  PROC DrawPart265()
    MoveL Offs(pOrigin,121.94,113.28,0.00),v40,z0,tPen\WObj:=wPaper;
    MoveL Offs(pOrigin,121.19,112.53,0.00),v40,z0,tPen\WObj:=wPaper;
    MoveL Offs(pOrigin,121.43,111.79,0.00),v40,z0,tPen\WObj:=wPaper;
    MoveL Offs(pOrigin,119.78,113.44,0.00),v40,z0,tPen\WObj:=wPaper;
    MoveL Offs(pOrigin,120.15,112.97,0.00),v40,z0,tPen\WObj:=wPaper;
    MoveL Offs(pOrigin,117.74,110.57,0.00),v40,z0,tPen\WObj:=wPaper;
    MoveL Offs(pOrigin,117.82,111.25,0.00),v40,z0,tPen\WObj:=wPaper;
    MoveL Offs(pOrigin,118.68,111.32,0.00),v40,z0,tPen\WObj:=wPaper;
    MoveL Offs(pOrigin,119.31,112.10,0.00),v40,z0,tPen\WObj:=wPaper;
    MoveL Offs(pOrigin,120.38,112.60,0.00),v40,z0,tPen\WObj:=wPaper;
    MoveL Offs(pOrigin,127.81,114.65,0.00),v40,fine,tPen\WObj:=wPaper;
    MoveL Offs(pOrigin,127.81,114.65,6.00),v60,z5,tPen\WObj:=wPaper;
    MoveL Offs(pOrigin,126.82,113.87,6.00),vTravel,z5,tPen\WObj:=wPaper;
    MoveL Offs(pOrigin,126.82,113.87,0.00),v60,z0,tPen\WObj:=wPaper;
    MoveL Offs(pOrigin,125.91,114.77,0.00),v40,fine,tPen\WObj:=wPaper;
    MoveL Offs(pOrigin,125.91,114.77,6.00),v60,z5,tPen\WObj:=wPaper;
    MoveL Offs(pOrigin,125.77,113.43,6.00),vTravel,z5,tPen\WObj:=wPaper;
    MoveL Offs(pOrigin,125.77,113.43,0.00),v60,z0,tPen\WObj:=wPaper;
    MoveL Offs(pOrigin,124.57,114.63,0.00),v40,fine,tPen\WObj:=wPaper;
    MoveL Offs(pOrigin,124.57,114.63,6.00),v60,z5,tPen\WObj:=wPaper;
    MoveL Offs(pOrigin,123.37,114.33,6.00),vTravel,z5,tPen\WObj:=wPaper;
    MoveL Offs(pOrigin,123.37,114.33,0.00),v60,z0,tPen\WObj:=wPaper;
    MoveL Offs(pOrigin,124.72,112.98,0.00),v40,fine,tPen\WObj:=wPaper;
    MoveL Offs(pOrigin,124.72,112.98,6.00),v60,z5,tPen\WObj:=wPaper;
    MoveL Offs(pOrigin,126.07,111.63,6.00),vTravel,z5,tPen\WObj:=wPaper;
    MoveL Offs(pOrigin,126.07,111.63,0.00),v60,z0,tPen\WObj:=wPaper;
    MoveL Offs(pOrigin,126.97,110.73,0.00),v40,fine,tPen\WObj:=wPaper;
    MoveL Offs(pOrigin,126.97,110.73,6.00),v60,z5,tPen\WObj:=wPaper;
    MoveL Offs(pOrigin,127.12,112.07,6.00),vTravel,z5,tPen\WObj:=wPaper;
    MoveL Offs(pOrigin,127.12,112.07,0.00),v60,z0,tPen\WObj:=wPaper;
    MoveL Offs(pOrigin,128.47,110.72,0.00),v40,fine,tPen\WObj:=wPaper;
    MoveL Offs(pOrigin,128.47,110.72,6.00),v60,z5,tPen\WObj:=wPaper;
    MoveL Offs(pOrigin,129.82,110.87,6.00),vTravel,z5,tPen\WObj:=wPaper;
    MoveL Offs(pOrigin,129.82,110.87,0.00),v60,z0,tPen\WObj:=wPaper;
    MoveL Offs(pOrigin,128.32,112.37,0.00),v40,fine,tPen\WObj:=wPaper;
    MoveL Offs(pOrigin,128.32,112.37,6.00),v60,z5,tPen\WObj:=wPaper;
    MoveL Offs(pOrigin,129.52,112.67,6.00),vTravel,z5,tPen\WObj:=wPaper;
    MoveL Offs(pOrigin,129.52,112.67,0.00),v60,z0,tPen\WObj:=wPaper;
    MoveL Offs(pOrigin,131.32,110.86,0.00),v40,fine,tPen\WObj:=wPaper;
    MoveL Offs(pOrigin,131.32,110.86,6.00),v60,z5,tPen\WObj:=wPaper;
    MoveL Offs(pOrigin,132.82,110.86,6.00),vTravel,z5,tPen\WObj:=wPaper;
    MoveL Offs(pOrigin,132.82,110.86,0.00),v60,z0,tPen\WObj:=wPaper;
    MoveL Offs(pOrigin,130.86,112.81,0.00),v40,fine,tPen\WObj:=wPaper;
    MoveL Offs(pOrigin,130.86,112.81,6.00),v60,z5,tPen\WObj:=wPaper;
    MoveL Offs(pOrigin,126.65,118.52,6.00),vTravel,z5,tPen\WObj:=wPaper;
    MoveL Offs(pOrigin,126.65,118.52,0.00),v60,z0,tPen\WObj:=wPaper;
    MoveL Offs(pOrigin,124.85,120.32,0.00),v40,z0,tPen\WObj:=wPaper;
    MoveL Offs(pOrigin,125.86,120.18,0.00),v40,z0,tPen\WObj:=wPaper;
    MoveL Offs(pOrigin,122.86,117.17,0.00),v40,z0,tPen\WObj:=wPaper;
    MoveL Offs(pOrigin,122.76,116.43,0.00),v40,z0,tPen\WObj:=wPaper;
    MoveL Offs(pOrigin,121.26,117.93,0.00),v40,z0,tPen\WObj:=wPaper;
    MoveL Offs(pOrigin,122.11,117.92,0.00),v40,z0,tPen\WObj:=wPaper;
    MoveL Offs(pOrigin,120.91,116.72,0.00),v40,z0,tPen\WObj:=wPaper;
    MoveL Offs(pOrigin,120.36,117.34,0.00),v40,z0,tPen\WObj:=wPaper;
    MoveL Offs(pOrigin,121.72,115.99,0.00),v40,z0,tPen\WObj:=wPaper;
    MoveL Offs(pOrigin,120.67,115.54,0.00),v40,z0,tPen\WObj:=wPaper;
    MoveL Offs(pOrigin,119.32,116.89,0.00),v40,z0,tPen\WObj:=wPaper;
    MoveL Offs(pOrigin,118.72,115.99,0.00),v40,z0,tPen\WObj:=wPaper;
    MoveL Offs(pOrigin,119.77,114.94,0.00),v40,fine,tPen\WObj:=wPaper;
    MoveL Offs(pOrigin,119.77,114.94,6.00),v60,z5,tPen\WObj:=wPaper;
    MoveL Offs(pOrigin,118.57,114.65,6.00),vTravel,z5,tPen\WObj:=wPaper;
    MoveL Offs(pOrigin,118.57,114.65,0.00),v60,z0,tPen\WObj:=wPaper;
    MoveL Offs(pOrigin,117.82,115.40,0.00),v40,fine,tPen\WObj:=wPaper;
    MoveL Offs(pOrigin,117.82,115.40,6.00),v60,z5,tPen\WObj:=wPaper;
    MoveL Offs(pOrigin,116.97,114.44,6.00),vTravel,z5,tPen\WObj:=wPaper;
    MoveL Offs(pOrigin,116.97,114.44,0.00),v60,z0,tPen\WObj:=wPaper;
    MoveL Offs(pOrigin,129.30,121.66,0.00),v40,z0,tPen\WObj:=wPaper;
    MoveL Offs(pOrigin,131.43,123.57,0.00),v40,z0,tPen\WObj:=wPaper;
    MoveL Offs(pOrigin,131.64,124.21,0.00),v40,fine,tPen\WObj:=wPaper;
    MoveL Offs(pOrigin,131.64,124.21,6.00),v60,z5,tPen\WObj:=wPaper;
    MoveL Offs(pOrigin,130.38,123.75,6.00),vTravel,z5,tPen\WObj:=wPaper;
    MoveL Offs(pOrigin,130.38,123.75,0.00),v60,z0,tPen\WObj:=wPaper;
    MoveL Offs(pOrigin,131.58,122.55,0.00),v40,z0,tPen\WObj:=wPaper;
    MoveL Offs(pOrigin,130.84,121.80,0.00),v40,z0,tPen\WObj:=wPaper;
    MoveL Offs(pOrigin,129.48,123.15,0.00),v40,z0,tPen\WObj:=wPaper;
    MoveL Offs(pOrigin,129.31,122.14,0.00),v40,z0,tPen\WObj:=wPaper;
    MoveL Offs(pOrigin,126.31,119.13,0.00),v40,fine,tPen\WObj:=wPaper;
    MoveL Offs(pOrigin,126.31,119.13,6.00),v60,z5,tPen\WObj:=wPaper;
    MoveL Offs(pOrigin,127.55,119.11,6.00),vTravel,z5,tPen\WObj:=wPaper;
    MoveL Offs(pOrigin,127.55,119.11,0.00),v60,z0,tPen\WObj:=wPaper;
    MoveL Offs(pOrigin,125.90,120.77,0.00),v40,z0,tPen\WObj:=wPaper;
    MoveL Offs(pOrigin,126.79,121.36,0.00),v40,z0,tPen\WObj:=wPaper;
    MoveL Offs(pOrigin,128.29,119.86,0.00),v40,z0,tPen\WObj:=wPaper;
    MoveL Offs(pOrigin,129.19,120.46,0.00),v40,z0,tPen\WObj:=wPaper;
    MoveL Offs(pOrigin,127.84,121.81,0.00),v40,z0,tPen\WObj:=wPaper;
    MoveL Offs(pOrigin,128.59,122.56,0.00),v40,z0,tPen\WObj:=wPaper;
    MoveL Offs(pOrigin,130.09,121.05,0.00),v40,fine,tPen\WObj:=wPaper;
    MoveL Offs(pOrigin,130.09,121.05,6.00),v60,z5,tPen\WObj:=wPaper;
    MoveL Offs(pOrigin,125.60,118.07,6.00),vTravel,z5,tPen\WObj:=wPaper;
    MoveL Offs(pOrigin,125.60,118.07,0.00),v60,z0,tPen\WObj:=wPaper;
    MoveL Offs(pOrigin,123.95,119.72,0.00),v40,z0,tPen\WObj:=wPaper;
    MoveL Offs(pOrigin,123.20,118.98,0.00),v40,z0,tPen\WObj:=wPaper;
    MoveL Offs(pOrigin,124.71,117.47,0.00),v40,z0,tPen\WObj:=wPaper;
    MoveL Offs(pOrigin,123.66,117.03,0.00),v40,z0,tPen\WObj:=wPaper;
    MoveL Offs(pOrigin,122.16,118.53,0.00),v40,fine,tPen\WObj:=wPaper;
    MoveL Offs(pOrigin,122.16,118.53,6.00),v60,z5,tPen\WObj:=wPaper;
    MoveL Offs(pOrigin,118.11,119.59,6.00),vTravel,z5,tPen\WObj:=wPaper;
    MoveL Offs(pOrigin,118.11,119.59,0.00),v60,z0,tPen\WObj:=wPaper;
    MoveL Offs(pOrigin,115.55,122.15,0.00),v40,z0,tPen\WObj:=wPaper;
    MoveL Offs(pOrigin,116.55,121.66,0.00),v40,z0,tPen\WObj:=wPaper;
    MoveL Offs(pOrigin,117.82,121.66,0.00),v40,z0,tPen\WObj:=wPaper;
    MoveL Offs(pOrigin,118.07,121.35,0.00),v40,z0,tPen\WObj:=wPaper;
    MoveL Offs(pOrigin,112.36,115.64,0.00),v40,z0,tPen\WObj:=wPaper;
    MoveL Offs(pOrigin,112.72,115.29,0.00),v40,z0,tPen\WObj:=wPaper;
    MoveL Offs(pOrigin,112.94,115.71,0.00),v40,z0,tPen\WObj:=wPaper;
    MoveL Offs(pOrigin,112.72,115.29,0.00),v40,z0,tPen\WObj:=wPaper;
    MoveL Offs(pOrigin,113.15,115.32,0.00),v40,z0,tPen\WObj:=wPaper;
    MoveL Offs(pOrigin,114.85,115.32,0.00),v40,z0,tPen\WObj:=wPaper;
    MoveL Offs(pOrigin,115.43,114.81,0.00),v40,z0,tPen\WObj:=wPaper;
    MoveL Offs(pOrigin,113.17,117.06,0.00),v40,z0,tPen\WObj:=wPaper;
    MoveL Offs(pOrigin,113.92,117.81,0.00),v40,z0,tPen\WObj:=wPaper;
    MoveL Offs(pOrigin,116.17,115.55,0.00),v40,z0,tPen\WObj:=wPaper;
    MoveL Offs(pOrigin,115.49,116.38,0.00),v40,z0,tPen\WObj:=wPaper;
    MoveL Offs(pOrigin,114.00,116.38,0.00),v40,fine,tPen\WObj:=wPaper;
    MoveL Offs(pOrigin,114.00,116.38,6.00),v60,z5,tPen\WObj:=wPaper;
    MoveL Offs(pOrigin,114.85,117.43,6.00),vTravel,z5,tPen\WObj:=wPaper;
    MoveL Offs(pOrigin,114.85,117.43,0.00),v60,z0,tPen\WObj:=wPaper;
    MoveL Offs(pOrigin,116.12,117.43,0.00),v40,fine,tPen\WObj:=wPaper;
    MoveL Offs(pOrigin,116.12,117.43,6.00),v60,z5,tPen\WObj:=wPaper;
    MoveL Offs(pOrigin,117.66,118.54,6.00),vTravel,z5,tPen\WObj:=wPaper;
  ENDPROC

  PROC DrawPart266()
    MoveL Offs(pOrigin,117.66,118.54,0.00),v60,z0,tPen\WObj:=wPaper;
    MoveL Offs(pOrigin,115.26,120.95,0.00),v40,z0,tPen\WObj:=wPaper;
    MoveL Offs(pOrigin,116.34,120.60,0.00),v40,z0,tPen\WObj:=wPaper;
    MoveL Offs(pOrigin,117.40,120.60,0.00),v40,z0,tPen\WObj:=wPaper;
    MoveL Offs(pOrigin,118.41,120.79,0.00),v40,z0,tPen\WObj:=wPaper;
    MoveL Offs(pOrigin,115.70,123.49,0.00),v40,fine,tPen\WObj:=wPaper;
    MoveL Offs(pOrigin,115.70,123.49,6.00),v60,z5,tPen\WObj:=wPaper;
    MoveL Offs(pOrigin,116.00,124.69,6.00),vTravel,z5,tPen\WObj:=wPaper;
    MoveL Offs(pOrigin,116.00,124.69,0.00),v60,z0,tPen\WObj:=wPaper;
    MoveL Offs(pOrigin,118.85,121.84,0.00),v40,fine,tPen\WObj:=wPaper;
    MoveL Offs(pOrigin,118.85,121.84,6.00),v60,z5,tPen\WObj:=wPaper;
    MoveL Offs(pOrigin,119.00,123.18,6.00),vTravel,z5,tPen\WObj:=wPaper;
    MoveL Offs(pOrigin,119.00,123.18,0.00),v60,z0,tPen\WObj:=wPaper;
    MoveL Offs(pOrigin,116.14,126.04,0.00),v40,z0,tPen\WObj:=wPaper;
    MoveL Offs(pOrigin,116.59,125.84,0.00),v40,z0,tPen\WObj:=wPaper;
    MoveL Offs(pOrigin,119.45,128.70,0.00),v40,z0,tPen\WObj:=wPaper;
    MoveL Offs(pOrigin,119.10,129.05,0.00),v40,z0,tPen\WObj:=wPaper;
    MoveL Offs(pOrigin,118.04,129.05,0.00),v40,z0,tPen\WObj:=wPaper;
    MoveL Offs(pOrigin,117.20,129.44,0.00),v40,z0,tPen\WObj:=wPaper;
    MoveL Offs(pOrigin,127.72,139.96,0.00),v40,z0,tPen\WObj:=wPaper;
    MoveL Offs(pOrigin,127.39,139.61,0.00),v40,z0,tPen\WObj:=wPaper;
    MoveL Offs(pOrigin,125.90,139.61,0.00),v40,fine,tPen\WObj:=wPaper;
    MoveL Offs(pOrigin,125.90,139.61,6.00),v60,z5,tPen\WObj:=wPaper;
    MoveL Offs(pOrigin,125.26,138.55,6.00),vTravel,z5,tPen\WObj:=wPaper;
    MoveL Offs(pOrigin,125.26,138.55,0.00),v60,z0,tPen\WObj:=wPaper;
    MoveL Offs(pOrigin,126.75,138.55,0.00),v40,fine,tPen\WObj:=wPaper;
    MoveL Offs(pOrigin,126.75,138.55,6.00),v60,z5,tPen\WObj:=wPaper;
    MoveL Offs(pOrigin,128.24,139.33,6.00),vTravel,z5,tPen\WObj:=wPaper;
    MoveL Offs(pOrigin,128.24,139.33,0.00),v60,z0,tPen\WObj:=wPaper;
    MoveL Offs(pOrigin,125.38,142.19,0.00),v40,fine,tPen\WObj:=wPaper;
    MoveL Offs(pOrigin,125.38,142.19,6.00),v60,z5,tPen\WObj:=wPaper;
    MoveL Offs(pOrigin,126.32,143.83,6.00),vTravel,z5,tPen\WObj:=wPaper;
    MoveL Offs(pOrigin,126.32,143.83,0.00),v60,z0,tPen\WObj:=wPaper;
    MoveL Offs(pOrigin,127.60,143.83,0.00),v40,z0,tPen\WObj:=wPaper;
    MoveL Offs(pOrigin,128.67,143.38,0.00),v40,z0,tPen\WObj:=wPaper;
    MoveL Offs(pOrigin,125.52,146.53,0.00),v40,fine,tPen\WObj:=wPaper;
    MoveL Offs(pOrigin,125.52,146.53,6.00),v60,z5,tPen\WObj:=wPaper;
    MoveL Offs(pOrigin,125.37,145.19,6.00),vTravel,z5,tPen\WObj:=wPaper;
    MoveL Offs(pOrigin,125.37,145.19,0.00),v60,z0,tPen\WObj:=wPaper;
    MoveL Offs(pOrigin,128.68,141.88,0.00),v40,fine,tPen\WObj:=wPaper;
    MoveL Offs(pOrigin,128.68,141.88,6.00),v60,z5,tPen\WObj:=wPaper;
    MoveL Offs(pOrigin,128.66,146.37,6.00),vTravel,z5,tPen\WObj:=wPaper;
    MoveL Offs(pOrigin,128.66,146.37,0.00),v60,z0,tPen\WObj:=wPaper;
    MoveL Offs(pOrigin,126.41,148.63,0.00),v40,z0,tPen\WObj:=wPaper;
    MoveL Offs(pOrigin,127.01,149.52,0.00),v40,z0,tPen\WObj:=wPaper;
    MoveL Offs(pOrigin,129.26,147.27,0.00),v40,z0,tPen\WObj:=wPaper;
    MoveL Offs(pOrigin,128.66,148.06,0.00),v40,z0,tPen\WObj:=wPaper;
    MoveL Offs(pOrigin,127.39,148.06,0.00),v40,fine,tPen\WObj:=wPaper;
    MoveL Offs(pOrigin,127.39,148.06,6.00),v60,z5,tPen\WObj:=wPaper;
    MoveL Offs(pOrigin,128.24,149.11,6.00),vTravel,z5,tPen\WObj:=wPaper;
    MoveL Offs(pOrigin,128.24,149.11,0.00),v60,z0,tPen\WObj:=wPaper;
    MoveL Offs(pOrigin,129.51,149.11,0.00),v40,z0,tPen\WObj:=wPaper;
    MoveL Offs(pOrigin,129.09,148.44,0.00),v40,z0,tPen\WObj:=wPaper;
    MoveL Offs(pOrigin,129.94,149.29,0.00),v40,z0,tPen\WObj:=wPaper;
    MoveL Offs(pOrigin,129.09,148.44,0.00),v40,z0,tPen\WObj:=wPaper;
    MoveL Offs(pOrigin,129.86,148.17,0.00),v40,z0,tPen\WObj:=wPaper;
    MoveL Offs(pOrigin,127.75,150.27,0.00),v40,z0,tPen\WObj:=wPaper;
    MoveL Offs(pOrigin,127.81,149.50,0.00),v40,z0,tPen\WObj:=wPaper;
    MoveL Offs(pOrigin,128.66,150.35,0.00),v40,z0,tPen\WObj:=wPaper;
    MoveL Offs(pOrigin,127.81,149.50,0.00),v40,fine,tPen\WObj:=wPaper;
    MoveL Offs(pOrigin,127.81,149.50,6.00),v60,z5,tPen\WObj:=wPaper;
    MoveL Offs(pOrigin,129.09,150.17,6.00),vTravel,z5,tPen\WObj:=wPaper;
    MoveL Offs(pOrigin,129.09,150.17,0.00),v60,z0,tPen\WObj:=wPaper;
    MoveL Offs(pOrigin,130.36,150.17,0.00),v40,z0,tPen\WObj:=wPaper;
    MoveL Offs(pOrigin,131.20,149.81,0.00),v40,z0,tPen\WObj:=wPaper;
    MoveL Offs(pOrigin,128.79,152.22,0.00),v40,z0,tPen\WObj:=wPaper;
    MoveL Offs(pOrigin,129.72,152.28,0.00),v40,z0,tPen\WObj:=wPaper;
    MoveL Offs(pOrigin,130.79,152.28,0.00),v40,z0,tPen\WObj:=wPaper;
    MoveL Offs(pOrigin,131.79,152.21,0.00),v40,z0,tPen\WObj:=wPaper;
    MoveL Offs(pOrigin,128.49,155.51,0.00),v40,fine,tPen\WObj:=wPaper;
    MoveL Offs(pOrigin,128.49,155.51,6.00),v60,z5,tPen\WObj:=wPaper;
    MoveL Offs(pOrigin,129.72,154.39,6.00),vTravel,z5,tPen\WObj:=wPaper;
    MoveL Offs(pOrigin,129.72,154.39,0.00),v60,z0,tPen\WObj:=wPaper;
    MoveL Offs(pOrigin,130.79,154.39,0.00),v40,fine,tPen\WObj:=wPaper;
    MoveL Offs(pOrigin,130.79,154.39,6.00),v60,z5,tPen\WObj:=wPaper;
    MoveL Offs(pOrigin,131.78,155.20,6.00),vTravel,z5,tPen\WObj:=wPaper;
    MoveL Offs(pOrigin,131.78,155.20,0.00),v60,z0,tPen\WObj:=wPaper;
    MoveL Offs(pOrigin,129.23,157.76,0.00),v40,z0,tPen\WObj:=wPaper;
    MoveL Offs(pOrigin,129.94,158.00,0.00),v40,z0,tPen\WObj:=wPaper;
    MoveL Offs(pOrigin,130.15,158.43,0.00),v40,z0,tPen\WObj:=wPaper;
    MoveL Offs(pOrigin,129.94,158.00,0.00),v40,fine,tPen\WObj:=wPaper;
    MoveL Offs(pOrigin,129.94,158.00,6.00),v60,z5,tPen\WObj:=wPaper;
    MoveL Offs(pOrigin,132.70,160.73,6.00),vTravel,z5,tPen\WObj:=wPaper;
    MoveL Offs(pOrigin,132.70,160.73,0.00),v60,z0,tPen\WObj:=wPaper;
    MoveL Offs(pOrigin,133.98,160.73,0.00),v40,fine,tPen\WObj:=wPaper;
    MoveL Offs(pOrigin,133.98,160.73,6.00),v60,z5,tPen\WObj:=wPaper;
    MoveL Offs(pOrigin,135.21,160.73,6.00),vTravel,z5,tPen\WObj:=wPaper;
    MoveL Offs(pOrigin,135.21,160.73,0.00),v60,z0,tPen\WObj:=wPaper;
    MoveL Offs(pOrigin,132.05,163.89,0.00),v40,z0,tPen\WObj:=wPaper;
    MoveL Offs(pOrigin,132.59,164.24,0.00),v40,z0,tPen\WObj:=wPaper;
    MoveL Offs(pOrigin,136.49,168.15,0.00),v40,z0,tPen\WObj:=wPaper;
    MoveL Offs(pOrigin,136.10,168.12,0.00),v40,z0,tPen\WObj:=wPaper;
    MoveL Offs(pOrigin,134.40,168.12,0.00),v40,z0,tPen\WObj:=wPaper;
    MoveL Offs(pOrigin,133.65,168.29,0.00),v40,z0,tPen\WObj:=wPaper;
    MoveL Offs(pOrigin,137.85,172.50,0.00),v40,z0,tPen\WObj:=wPaper;
    MoveL Offs(pOrigin,138.47,172.41,0.00),v40,z0,tPen\WObj:=wPaper;
    MoveL Offs(pOrigin,135.77,175.11,0.00),v40,z0,tPen\WObj:=wPaper;
    MoveL Offs(pOrigin,136.22,175.34,0.00),v40,z0,tPen\WObj:=wPaper;
    MoveL Offs(pOrigin,138.92,178.04,0.00),v40,z0,tPen\WObj:=wPaper;
    MoveL Offs(pOrigin,139.20,177.65,0.00),v40,z0,tPen\WObj:=wPaper;
    MoveL Offs(pOrigin,136.80,180.05,0.00),v40,fine,tPen\WObj:=wPaper;
    MoveL Offs(pOrigin,136.80,180.05,6.00),v60,z5,tPen\WObj:=wPaper;
    MoveL Offs(pOrigin,137.09,181.25,6.00),vTravel,z5,tPen\WObj:=wPaper;
    MoveL Offs(pOrigin,137.09,181.25,0.00),v60,z0,tPen\WObj:=wPaper;
    MoveL Offs(pOrigin,139.50,178.85,0.00),v40,fine,tPen\WObj:=wPaper;
    MoveL Offs(pOrigin,139.50,178.85,6.00),v60,z5,tPen\WObj:=wPaper;
    MoveL Offs(pOrigin,137.58,181.18,6.00),vTravel,z5,tPen\WObj:=wPaper;
    MoveL Offs(pOrigin,137.58,181.18,0.00),v60,z0,tPen\WObj:=wPaper;
    MoveL Offs(pOrigin,145.70,189.30,0.00),v40,z0,tPen\WObj:=wPaper;
    MoveL Offs(pOrigin,145.16,189.61,0.00),v40,z0,tPen\WObj:=wPaper;
    MoveL Offs(pOrigin,147.56,187.21,0.00),v40,z0,tPen\WObj:=wPaper;
    MoveL Offs(pOrigin,148.61,187.66,0.00),v40,z0,tPen\WObj:=wPaper;
    MoveL Offs(pOrigin,146.21,190.06,0.00),v40,fine,tPen\WObj:=wPaper;
    MoveL Offs(pOrigin,146.21,190.06,6.00),v60,z5,tPen\WObj:=wPaper;
    MoveL Offs(pOrigin,144.11,189.17,6.00),vTravel,z5,tPen\WObj:=wPaper;
    MoveL Offs(pOrigin,144.11,189.17,0.00),v60,z0,tPen\WObj:=wPaper;
    MoveL Offs(pOrigin,146.51,186.76,0.00),v40,z0,tPen\WObj:=wPaper;
    MoveL Offs(pOrigin,146.07,185.72,0.00),v40,z0,tPen\WObj:=wPaper;
    MoveL Offs(pOrigin,143.06,188.72,0.00),v40,z0,tPen\WObj:=wPaper;
    MoveL Offs(pOrigin,142.02,188.28,0.00),v40,z0,tPen\WObj:=wPaper;
  ENDPROC

  PROC DrawPart267()
    MoveL Offs(pOrigin,146.07,184.22,0.00),v40,z0,tPen\WObj:=wPaper;
    MoveL Offs(pOrigin,145.38,184.50,0.00),v40,z0,tPen\WObj:=wPaper;
    MoveL Offs(pOrigin,144.18,183.30,0.00),v40,z0,tPen\WObj:=wPaper;
    MoveL Offs(pOrigin,143.38,183.93,0.00),v40,z0,tPen\WObj:=wPaper;
    MoveL Offs(pOrigin,146.23,181.07,0.00),v40,z0,tPen\WObj:=wPaper;
    MoveL Offs(pOrigin,145.82,180.46,0.00),v40,z0,tPen\WObj:=wPaper;
    MoveL Offs(pOrigin,144.32,178.96,0.00),v40,z0,tPen\WObj:=wPaper;
    MoveL Offs(pOrigin,143.69,179.13,0.00),v40,z0,tPen\WObj:=wPaper;
    MoveL Offs(pOrigin,147.30,175.53,0.00),v40,z0,tPen\WObj:=wPaper;
    MoveL Offs(pOrigin,146.70,175.37,0.00),v40,z0,tPen\WObj:=wPaper;
    MoveL Offs(pOrigin,145.35,174.02,0.00),v40,z0,tPen\WObj:=wPaper;
    MoveL Offs(pOrigin,144.76,173.59,0.00),v40,z0,tPen\WObj:=wPaper;
    MoveL Offs(pOrigin,148.81,169.53,0.00),v40,z0,tPen\WObj:=wPaper;
    MoveL Offs(pOrigin,148.33,169.53,0.00),v40,z0,tPen\WObj:=wPaper;
    MoveL Offs(pOrigin,146.83,168.03,0.00),v40,z0,tPen\WObj:=wPaper;
    MoveL Offs(pOrigin,146.38,169.08,0.00),v40,z0,tPen\WObj:=wPaper;
    MoveL Offs(pOrigin,147.89,170.58,0.00),v40,z0,tPen\WObj:=wPaper;
    MoveL Offs(pOrigin,148.21,171.63,0.00),v40,z0,tPen\WObj:=wPaper;
    MoveL Offs(pOrigin,144.30,175.54,0.00),v40,z0,tPen\WObj:=wPaper;
    MoveL Offs(pOrigin,144.90,175.06,0.00),v40,z0,tPen\WObj:=wPaper;
    MoveL Offs(pOrigin,146.41,176.57,0.00),v40,z0,tPen\WObj:=wPaper;
    MoveL Offs(pOrigin,146.84,177.48,0.00),v40,z0,tPen\WObj:=wPaper;
    MoveL Offs(pOrigin,143.39,180.93,0.00),v40,z0,tPen\WObj:=wPaper;
    MoveL Offs(pOrigin,144.17,180.31,0.00),v40,z0,tPen\WObj:=wPaper;
    MoveL Offs(pOrigin,145.67,181.81,0.00),v40,z0,tPen\WObj:=wPaper;
    MoveL Offs(pOrigin,146.08,182.72,0.00),v40,z0,tPen\WObj:=wPaper;
    MoveL Offs(pOrigin,141.12,187.68,0.00),v40,z0,tPen\WObj:=wPaper;
    MoveL Offs(pOrigin,142.05,187.75,0.00),v40,z0,tPen\WObj:=wPaper;
    MoveL Offs(pOrigin,142.48,187.96,0.00),v40,z0,tPen\WObj:=wPaper;
    MoveL Offs(pOrigin,142.05,187.75,0.00),v40,fine,tPen\WObj:=wPaper;
    MoveL Offs(pOrigin,142.05,187.75,6.00),v60,z5,tPen\WObj:=wPaper;
    MoveL Offs(pOrigin,139.63,186.19,6.00),vTravel,z5,tPen\WObj:=wPaper;
    MoveL Offs(pOrigin,139.63,186.19,0.00),v60,z0,tPen\WObj:=wPaper;
    MoveL Offs(pOrigin,141.73,184.08,0.00),v40,fine,tPen\WObj:=wPaper;
    MoveL Offs(pOrigin,141.73,184.08,6.00),v60,z5,tPen\WObj:=wPaper;
    MoveL Offs(pOrigin,140.69,182.14,6.00),vTravel,z5,tPen\WObj:=wPaper;
    MoveL Offs(pOrigin,140.69,182.14,0.00),v60,z0,tPen\WObj:=wPaper;
    MoveL Offs(pOrigin,138.28,184.54,0.00),v40,fine,tPen\WObj:=wPaper;
    MoveL Offs(pOrigin,138.28,184.54,6.00),v60,z5,tPen\WObj:=wPaper;
    MoveL Offs(pOrigin,143.38,182.43,6.00),vTravel,z5,tPen\WObj:=wPaper;
    MoveL Offs(pOrigin,143.38,182.43,0.00),v60,z0,tPen\WObj:=wPaper;
    MoveL Offs(pOrigin,146.39,179.42,0.00),v40,z0,tPen\WObj:=wPaper;
    MoveL Offs(pOrigin,146.11,179.26,0.00),v40,z0,tPen\WObj:=wPaper;
    MoveL Offs(pOrigin,144.46,177.61,0.00),v40,z0,tPen\WObj:=wPaper;
    MoveL Offs(pOrigin,143.85,177.49,0.00),v40,z0,tPen\WObj:=wPaper;
    MoveL Offs(pOrigin,147.75,173.58,0.00),v40,z0,tPen\WObj:=wPaper;
    MoveL Offs(pOrigin,147.29,172.97,0.00),v40,z0,tPen\WObj:=wPaper;
    MoveL Offs(pOrigin,145.79,171.47,0.00),v40,z0,tPen\WObj:=wPaper;
    MoveL Offs(pOrigin,145.21,171.64,0.00),v40,z0,tPen\WObj:=wPaper;
    MoveL Offs(pOrigin,149.42,167.43,0.00),v40,z0,tPen\WObj:=wPaper;
    MoveL Offs(pOrigin,148.92,167.14,0.00),v40,z0,tPen\WObj:=wPaper;
    MoveL Offs(pOrigin,146.37,164.58,0.00),v40,z0,tPen\WObj:=wPaper;
    MoveL Offs(pOrigin,146.30,164.38,0.00),v40,z0,tPen\WObj:=wPaper;
    MoveL Offs(pOrigin,146.09,164.80,0.00),v40,z0,tPen\WObj:=wPaper;
    MoveL Offs(pOrigin,146.30,164.38,0.00),v40,z0,tPen\WObj:=wPaper;
    MoveL Offs(pOrigin,146.73,163.52,0.00),v40,z0,tPen\WObj:=wPaper;
    MoveL Offs(pOrigin,146.51,163.95,0.00),v40,z0,tPen\WObj:=wPaper;
    MoveL Offs(pOrigin,146.73,163.52,0.00),v40,z0,tPen\WObj:=wPaper;
    MoveL Offs(pOrigin,146.67,163.39,0.00),v40,z0,tPen\WObj:=wPaper;
    MoveL Offs(pOrigin,149.22,165.94,0.00),v40,z0,tPen\WObj:=wPaper;
    MoveL Offs(pOrigin,149.67,164.89,0.00),v40,z0,tPen\WObj:=wPaper;
    MoveL Offs(pOrigin,147.11,162.34,0.00),v40,z0,tPen\WObj:=wPaper;
    MoveL Offs(pOrigin,147.36,162.46,0.00),v40,z0,tPen\WObj:=wPaper;
    MoveL Offs(pOrigin,147.15,162.89,0.00),v40,z0,tPen\WObj:=wPaper;
    MoveL Offs(pOrigin,147.36,162.46,0.00),v40,z0,tPen\WObj:=wPaper;
    MoveL Offs(pOrigin,148.21,161.82,0.00),v40,z0,tPen\WObj:=wPaper;
    MoveL Offs(pOrigin,146.87,163.52,0.00),v40,z0,tPen\WObj:=wPaper;
    MoveL Offs(pOrigin,144.53,167.99,0.00),v40,z0,tPen\WObj:=wPaper;
    MoveL Offs(pOrigin,142.26,173.73,0.00),v40,fine,tPen\WObj:=wPaper;
    MoveL Offs(pOrigin,142.26,173.73,6.00),v60,z5,tPen\WObj:=wPaper;
    MoveL Offs(pOrigin,142.82,171.05,6.00),vTravel,z5,tPen\WObj:=wPaper;
    MoveL Offs(pOrigin,142.82,171.05,0.00),v60,z0,tPen\WObj:=wPaper;
    MoveL Offs(pOrigin,150.93,162.93,0.00),v40,z0,tPen\WObj:=wPaper;
    MoveL Offs(pOrigin,150.41,162.65,0.00),v40,z0,tPen\WObj:=wPaper;
    MoveL Offs(pOrigin,148.00,160.24,0.00),v40,z0,tPen\WObj:=wPaper;
    MoveL Offs(pOrigin,148.64,160.73,0.00),v40,z0,tPen\WObj:=wPaper;
    MoveL Offs(pOrigin,150.55,160.73,0.00),v40,z0,tPen\WObj:=wPaper;
    MoveL Offs(pOrigin,151.15,160.40,0.00),v40,z0,tPen\WObj:=wPaper;
    MoveL Offs(pOrigin,149.05,158.30,0.00),v40,z0,tPen\WObj:=wPaper;
    MoveL Offs(pOrigin,149.49,158.62,0.00),v40,z0,tPen\WObj:=wPaper;
    MoveL Offs(pOrigin,151.19,158.62,0.00),v40,z0,tPen\WObj:=wPaper;
    MoveL Offs(pOrigin,151.45,159.21,0.00),v40,z0,tPen\WObj:=wPaper;
    MoveL Offs(pOrigin,149.49,157.25,0.00),v40,z0,tPen\WObj:=wPaper;
    MoveL Offs(pOrigin,149.91,157.15,0.00),v40,z0,tPen\WObj:=wPaper;
    MoveL Offs(pOrigin,149.70,157.57,0.00),v40,z0,tPen\WObj:=wPaper;
    MoveL Offs(pOrigin,149.91,157.15,0.00),v40,z0,tPen\WObj:=wPaper;
    MoveL Offs(pOrigin,149.91,157.56,0.00),v40,z0,tPen\WObj:=wPaper;
    MoveL Offs(pOrigin,151.61,157.56,0.00),v40,z0,tPen\WObj:=wPaper;
    MoveL Offs(pOrigin,151.74,158.01,0.00),v40,z0,tPen\WObj:=wPaper;
    MoveL Offs(pOrigin,149.94,156.21,0.00),v40,z0,tPen\WObj:=wPaper;
    MoveL Offs(pOrigin,150.55,156.09,0.00),v40,z0,tPen\WObj:=wPaper;
    MoveL Offs(pOrigin,150.34,156.51,0.00),v40,z0,tPen\WObj:=wPaper;
    MoveL Offs(pOrigin,150.55,156.09,0.00),v40,z0,tPen\WObj:=wPaper;
    MoveL Offs(pOrigin,150.55,156.50,0.00),v40,z0,tPen\WObj:=wPaper;
    MoveL Offs(pOrigin,151.82,156.50,0.00),v40,z0,tPen\WObj:=wPaper;
    MoveL Offs(pOrigin,152.19,156.96,0.00),v40,z0,tPen\WObj:=wPaper;
    MoveL Offs(pOrigin,150.54,155.31,0.00),v40,z0,tPen\WObj:=wPaper;
    MoveL Offs(pOrigin,150.98,155.45,0.00),v40,z0,tPen\WObj:=wPaper;
    MoveL Offs(pOrigin,152.25,155.45,0.00),v40,z0,tPen\WObj:=wPaper;
    MoveL Offs(pOrigin,152.48,155.76,0.00),v40,z0,tPen\WObj:=wPaper;
    MoveL Offs(pOrigin,150.83,154.11,0.00),v40,z0,tPen\WObj:=wPaper;
    MoveL Offs(pOrigin,151.40,154.39,0.00),v40,z0,tPen\WObj:=wPaper;
    MoveL Offs(pOrigin,152.46,154.39,0.00),v40,z0,tPen\WObj:=wPaper;
    MoveL Offs(pOrigin,152.93,154.72,0.00),v40,z0,tPen\WObj:=wPaper;
    MoveL Offs(pOrigin,151.28,153.06,0.00),v40,z0,tPen\WObj:=wPaper;
    MoveL Offs(pOrigin,151.61,153.34,0.00),v40,z0,tPen\WObj:=wPaper;
    MoveL Offs(pOrigin,152.68,153.34,0.00),v40,z0,tPen\WObj:=wPaper;
    MoveL Offs(pOrigin,153.38,153.67,0.00),v40,z0,tPen\WObj:=wPaper;
    MoveL Offs(pOrigin,151.57,151.87,0.00),v40,z0,tPen\WObj:=wPaper;
    MoveL Offs(pOrigin,152.04,152.28,0.00),v40,z0,tPen\WObj:=wPaper;
    MoveL Offs(pOrigin,153.10,152.28,0.00),v40,z0,tPen\WObj:=wPaper;
    MoveL Offs(pOrigin,153.67,152.47,0.00),v40,z0,tPen\WObj:=wPaper;
    MoveL Offs(pOrigin,152.02,150.82,0.00),v40,z0,tPen\WObj:=wPaper;
    MoveL Offs(pOrigin,151.42,150.50,0.00),v40,z0,tPen\WObj:=wPaper;
    MoveL Offs(pOrigin,156.38,145.54,0.00),v40,z0,tPen\WObj:=wPaper;
    MoveL Offs(pOrigin,155.90,145.74,0.00),v40,z0,tPen\WObj:=wPaper;
    MoveL Offs(pOrigin,154.10,143.93,0.00),v40,z0,tPen\WObj:=wPaper;
    MoveL Offs(pOrigin,154.80,143.83,0.00),v40,z0,tPen\WObj:=wPaper;
    MoveL Offs(pOrigin,155.86,143.83,0.00),v40,z0,tPen\WObj:=wPaper;
    MoveL Offs(pOrigin,156.19,144.54,0.00),v40,z0,tPen\WObj:=wPaper;
  ENDPROC

  PROC DrawPart268()
    MoveL Offs(pOrigin,154.54,142.89,0.00),v40,z0,tPen\WObj:=wPaper;
    MoveL Offs(pOrigin,155.01,142.78,0.00),v40,z0,tPen\WObj:=wPaper;
    MoveL Offs(pOrigin,156.07,142.78,0.00),v40,z0,tPen\WObj:=wPaper;
    MoveL Offs(pOrigin,156.49,143.34,0.00),v40,z0,tPen\WObj:=wPaper;
    MoveL Offs(pOrigin,154.84,141.69,0.00),v40,z0,tPen\WObj:=wPaper;
    MoveL Offs(pOrigin,155.44,141.72,0.00),v40,z0,tPen\WObj:=wPaper;
    MoveL Offs(pOrigin,156.50,141.72,0.00),v40,z0,tPen\WObj:=wPaper;
    MoveL Offs(pOrigin,156.94,142.30,0.00),v40,z0,tPen\WObj:=wPaper;
    MoveL Offs(pOrigin,151.98,137.34,0.00),v40,z0,tPen\WObj:=wPaper;
    MoveL Offs(pOrigin,152.72,136.59,0.00),v40,z0,tPen\WObj:=wPaper;
    MoveL Offs(pOrigin,157.23,141.10,0.00),v40,z0,tPen\WObj:=wPaper;
    MoveL Offs(pOrigin,156.93,140.66,0.00),v40,z0,tPen\WObj:=wPaper;
    MoveL Offs(pOrigin,155.65,140.66,0.00),v40,z0,tPen\WObj:=wPaper;
    MoveL Offs(pOrigin,156.07,139.61,0.00),v40,z0,tPen\WObj:=wPaper;
    MoveL Offs(pOrigin,157.14,139.61,0.00),v40,z0,tPen\WObj:=wPaper;
    MoveL Offs(pOrigin,157.53,139.90,0.00),v40,z0,tPen\WObj:=wPaper;
    MoveL Offs(pOrigin,153.62,135.99,0.00),v40,z0,tPen\WObj:=wPaper;
    MoveL Offs(pOrigin,153.74,136.44,0.00),v40,z0,tPen\WObj:=wPaper;
    MoveL Offs(pOrigin,158.20,136.44,0.00),v40,z0,tPen\WObj:=wPaper;
    MoveL Offs(pOrigin,158.57,136.46,0.00),v40,z0,tPen\WObj:=wPaper;
    MoveL Offs(pOrigin,155.71,133.60,0.00),v40,z0,tPen\WObj:=wPaper;
    MoveL Offs(pOrigin,156.30,133.99,0.00),v40,z0,tPen\WObj:=wPaper;
    MoveL Offs(pOrigin,156.30,137.39,0.00),v40,z0,tPen\WObj:=wPaper;
    MoveL Offs(pOrigin,155.25,137.60,0.00),v40,z0,tPen\WObj:=wPaper;
    MoveL Offs(pOrigin,155.25,135.26,0.00),v40,z0,tPen\WObj:=wPaper;
    MoveL Offs(pOrigin,154.59,135.38,0.00),v40,z0,tPen\WObj:=wPaper;
    MoveL Offs(pOrigin,158.41,135.38,0.00),v40,z0,tPen\WObj:=wPaper;
    MoveL Offs(pOrigin,158.84,134.33,0.00),v40,z0,tPen\WObj:=wPaper;
    MoveL Offs(pOrigin,155.65,134.33,0.00),v40,z0,tPen\WObj:=wPaper;
    MoveL Offs(pOrigin,155.12,134.50,0.00),v40,z0,tPen\WObj:=wPaper;
    MoveL Offs(pOrigin,158.12,137.51,0.00),v40,z0,tPen\WObj:=wPaper;
    MoveL Offs(pOrigin,158.80,137.14,0.00),v40,z0,tPen\WObj:=wPaper;
    MoveL Offs(pOrigin,153.84,142.10,0.00),v40,z0,tPen\WObj:=wPaper;
    MoveL Offs(pOrigin,153.19,141.54,0.00),v40,z0,tPen\WObj:=wPaper;
    MoveL Offs(pOrigin,150.33,138.68,0.00),v40,z0,tPen\WObj:=wPaper;
    MoveL Offs(pOrigin,150.98,138.66,0.00),v40,z0,tPen\WObj:=wPaper;
    MoveL Offs(pOrigin,144.81,142.77,0.00),v40,z0,tPen\WObj:=wPaper;
    MoveL Offs(pOrigin,139.29,145.25,0.00),v40,fine,tPen\WObj:=wPaper;
    MoveL Offs(pOrigin,139.29,145.25,6.00),v60,z5,tPen\WObj:=wPaper;
    MoveL Offs(pOrigin,140.65,144.84,6.00),vTravel,z5,tPen\WObj:=wPaper;
    MoveL Offs(pOrigin,140.65,144.84,0.00),v60,z0,tPen\WObj:=wPaper;
    MoveL Offs(pOrigin,143.36,142.13,0.00),v40,fine,tPen\WObj:=wPaper;
    MoveL Offs(pOrigin,143.36,142.13,6.00),v60,z5,tPen\WObj:=wPaper;
    MoveL Offs(pOrigin,144.55,143.93,6.00),vTravel,z5,tPen\WObj:=wPaper;
    MoveL Offs(pOrigin,144.55,143.93,0.00),v60,z0,tPen\WObj:=wPaper;
    MoveL Offs(pOrigin,161.08,127.40,0.00),v40,fine,tPen\WObj:=wPaper;
    MoveL Offs(pOrigin,161.08,127.40,6.00),v60,z5,tPen\WObj:=wPaper;
    MoveL Offs(pOrigin,160.54,125.88,6.00),vTravel,z5,tPen\WObj:=wPaper;
    MoveL Offs(pOrigin,160.54,125.88,0.00),v60,z0,tPen\WObj:=wPaper;
    MoveL Offs(pOrigin,156.07,125.88,0.00),v40,z0,tPen\WObj:=wPaper;
    MoveL Offs(pOrigin,156.07,126.94,0.00),v40,z0,tPen\WObj:=wPaper;
    MoveL Offs(pOrigin,154.80,126.94,0.00),v40,fine,tPen\WObj:=wPaper;
    MoveL Offs(pOrigin,154.80,126.94,6.00),v60,z5,tPen\WObj:=wPaper;
    MoveL Offs(pOrigin,155.10,130.01,6.00),vTravel,z5,tPen\WObj:=wPaper;
    MoveL Offs(pOrigin,155.10,130.01,0.00),v60,z0,tPen\WObj:=wPaper;
    MoveL Offs(pOrigin,159.16,134.06,0.00),v40,z0,tPen\WObj:=wPaper;
    MoveL Offs(pOrigin,158.41,133.56,0.00),v40,z0,tPen\WObj:=wPaper;
    MoveL Offs(pOrigin,158.41,131.44,0.00),v40,z0,tPen\WObj:=wPaper;
    MoveL Offs(pOrigin,157.99,131.16,0.00),v40,z0,tPen\WObj:=wPaper;
    MoveL Offs(pOrigin,159.48,131.16,0.00),v40,z0,tPen\WObj:=wPaper;
    MoveL Offs(pOrigin,160.47,131.00,0.00),v40,z0,tPen\WObj:=wPaper;
    MoveL Offs(pOrigin,136.13,155.34,0.00),v40,fine,tPen\WObj:=wPaper;
    MoveL Offs(pOrigin,136.13,155.34,6.00),v60,z5,tPen\WObj:=wPaper;
    MoveL Offs(pOrigin,137.16,154.39,6.00),vTravel,z5,tPen\WObj:=wPaper;
    MoveL Offs(pOrigin,137.16,154.39,0.00),v60,z0,tPen\WObj:=wPaper;
    MoveL Offs(pOrigin,137.16,153.96,0.00),v40,z0,tPen\WObj:=wPaper;
    MoveL Offs(pOrigin,138.01,153.32,0.00),v40,z0,tPen\WObj:=wPaper;
    MoveL Offs(pOrigin,137.80,153.32,0.00),v40,z0,tPen\WObj:=wPaper;
    MoveL Offs(pOrigin,137.05,153.77,0.00),v40,z0,tPen\WObj:=wPaper;
    MoveL Offs(pOrigin,137.95,154.67,0.00),v40,z0,tPen\WObj:=wPaper;
    MoveL Offs(pOrigin,137.77,155.18,0.00),v40,z0,tPen\WObj:=wPaper;
    MoveL Offs(pOrigin,160.01,132.95,0.00),v40,fine,tPen\WObj:=wPaper;
    MoveL Offs(pOrigin,160.01,132.95,6.00),v60,z5,tPen\WObj:=wPaper;
    MoveL Offs(pOrigin,156.93,132.93,6.00),vTravel,z5,tPen\WObj:=wPaper;
    MoveL Offs(pOrigin,156.93,132.93,0.00),v60,z0,tPen\WObj:=wPaper;
    MoveL Offs(pOrigin,155.01,134.84,0.00),v40,z0,tPen\WObj:=wPaper;
    MoveL Offs(pOrigin,156.93,132.93,0.00),v40,fine,tPen\WObj:=wPaper;
    MoveL Offs(pOrigin,156.93,132.93,6.00),v60,z5,tPen\WObj:=wPaper;
    MoveL Offs(pOrigin,155.56,131.96,6.00),vTravel,z5,tPen\WObj:=wPaper;
    MoveL Offs(pOrigin,155.56,131.96,0.00),v60,z0,tPen\WObj:=wPaper;
    MoveL Offs(pOrigin,154.20,130.60,0.00),v40,z0,tPen\WObj:=wPaper;
    MoveL Offs(pOrigin,154.38,131.16,0.00),v40,z0,tPen\WObj:=wPaper;
    MoveL Offs(pOrigin,155.44,131.16,0.00),v40,z0,tPen\WObj:=wPaper;
    MoveL Offs(pOrigin,154.80,130.59,0.00),v40,z0,tPen\WObj:=wPaper;
    MoveL Offs(pOrigin,155.51,130.02,0.00),v40,z0,tPen\WObj:=wPaper;
    MoveL Offs(pOrigin,152.04,132.57,0.00),v40,z0,tPen\WObj:=wPaper;
    MoveL Offs(pOrigin,148.21,134.48,0.00),v40,z0,tPen\WObj:=wPaper;
    MoveL Offs(pOrigin,144.18,135.97,0.00),v40,z0,tPen\WObj:=wPaper;
    MoveL Offs(pOrigin,143.75,136.75,0.00),v40,z0,tPen\WObj:=wPaper;
    MoveL Offs(pOrigin,143.75,136.75,0.00),v40,z0,tPen\WObj:=wPaper;
    MoveL Offs(pOrigin,148.00,135.55,0.00),v40,z0,tPen\WObj:=wPaper;
    MoveL Offs(pOrigin,151.40,134.06,0.00),v40,z0,tPen\WObj:=wPaper;
    MoveL Offs(pOrigin,156.78,130.45,0.00),v40,z0,tPen\WObj:=wPaper;
    MoveL Offs(pOrigin,156.29,130.80,0.00),v40,fine,tPen\WObj:=wPaper;
    MoveL Offs(pOrigin,156.29,130.80,6.00),v60,z5,tPen\WObj:=wPaper;
    MoveL Offs(pOrigin,154.51,132.40,6.00),vTravel,z5,tPen\WObj:=wPaper;
    MoveL Offs(pOrigin,154.51,132.40,0.00),v60,z0,tPen\WObj:=wPaper;
    MoveL Offs(pOrigin,153.31,131.20,0.00),v40,z0,tPen\WObj:=wPaper;
    MoveL Offs(pOrigin,152.56,131.95,0.00),v40,z0,tPen\WObj:=wPaper;
    MoveL Offs(pOrigin,153.61,133.00,0.00),v40,z0,tPen\WObj:=wPaper;
    MoveL Offs(pOrigin,152.72,133.59,0.00),v40,z0,tPen\WObj:=wPaper;
    MoveL Offs(pOrigin,151.51,132.39,0.00),v40,z0,tPen\WObj:=wPaper;
    MoveL Offs(pOrigin,150.62,132.99,0.00),v40,z0,tPen\WObj:=wPaper;
    MoveL Offs(pOrigin,151.82,134.19,0.00),v40,z0,tPen\WObj:=wPaper;
    MoveL Offs(pOrigin,152.82,134.17,0.00),v40,z0,tPen\WObj:=wPaper;
    MoveL Offs(pOrigin,161.23,125.75,0.00),v40,fine,tPen\WObj:=wPaper;
    MoveL Offs(pOrigin,161.23,125.75,6.00),v60,z5,tPen\WObj:=wPaper;
    MoveL Offs(pOrigin,161.69,123.80,6.00),vTravel,z5,tPen\WObj:=wPaper;
    MoveL Offs(pOrigin,161.69,123.80,0.00),v60,z0,tPen\WObj:=wPaper;
    MoveL Offs(pOrigin,149.82,135.67,0.00),v40,z0,tPen\WObj:=wPaper;
    MoveL Offs(pOrigin,149.72,135.08,0.00),v40,z0,tPen\WObj:=wPaper;
    MoveL Offs(pOrigin,148.52,133.88,0.00),v40,z0,tPen\WObj:=wPaper;
    MoveL Offs(pOrigin,147.58,133.43,0.00),v40,z0,tPen\WObj:=wPaper;
    MoveL Offs(pOrigin,143.22,137.79,0.00),v40,fine,tPen\WObj:=wPaper;
    MoveL Offs(pOrigin,143.22,137.79,6.00),v60,z5,tPen\WObj:=wPaper;
    MoveL Offs(pOrigin,145.38,135.22,6.00),vTravel,z5,tPen\WObj:=wPaper;
    MoveL Offs(pOrigin,145.38,135.22,0.00),v60,z0,tPen\WObj:=wPaper;
    MoveL Offs(pOrigin,146.58,136.42,0.00),v40,z0,tPen\WObj:=wPaper;
    MoveL Offs(pOrigin,147.57,136.43,0.00),v40,z0,tPen\WObj:=wPaper;
    MoveL Offs(pOrigin,161.99,122.00,0.00),v40,fine,tPen\WObj:=wPaper;
  ENDPROC

  PROC DrawPart269()
    MoveL Offs(pOrigin,161.99,122.00,6.00),v60,z5,tPen\WObj:=wPaper;
    MoveL Offs(pOrigin,161.39,120.60,6.00),vTravel,z5,tPen\WObj:=wPaper;
    MoveL Offs(pOrigin,161.39,120.60,0.00),v60,z0,tPen\WObj:=wPaper;
    MoveL Offs(pOrigin,159.90,120.60,0.00),v40,z0,tPen\WObj:=wPaper;
    MoveL Offs(pOrigin,160.53,121.24,0.00),v40,z0,tPen\WObj:=wPaper;
    MoveL Offs(pOrigin,160.53,123.58,0.00),v40,fine,tPen\WObj:=wPaper;
    MoveL Offs(pOrigin,160.53,123.58,6.00),v60,z5,tPen\WObj:=wPaper;
    MoveL Offs(pOrigin,159.47,122.94,6.00),vTravel,z5,tPen\WObj:=wPaper;
    MoveL Offs(pOrigin,159.47,122.94,0.00),v60,z0,tPen\WObj:=wPaper;
    MoveL Offs(pOrigin,159.47,129.31,0.00),v40,fine,tPen\WObj:=wPaper;
    MoveL Offs(pOrigin,159.47,129.31,6.00),v60,z5,tPen\WObj:=wPaper;
    MoveL Offs(pOrigin,160.92,129.05,6.00),vTravel,z5,tPen\WObj:=wPaper;
    MoveL Offs(pOrigin,160.92,129.05,0.00),v60,z0,tPen\WObj:=wPaper;
    MoveL Offs(pOrigin,147.55,142.42,0.00),v40,fine,tPen\WObj:=wPaper;
    MoveL Offs(pOrigin,147.55,142.42,6.00),v60,z5,tPen\WObj:=wPaper;
    MoveL Offs(pOrigin,148.85,143.17,6.00),vTravel,z5,tPen\WObj:=wPaper;
    MoveL Offs(pOrigin,148.85,143.17,0.00),v60,z0,tPen\WObj:=wPaper;
    MoveL Offs(pOrigin,150.35,144.67,0.00),v40,z0,tPen\WObj:=wPaper;
    MoveL Offs(pOrigin,150.12,144.40,0.00),v40,z0,tPen\WObj:=wPaper;
    MoveL Offs(pOrigin,150.34,143.98,0.00),v40,z0,tPen\WObj:=wPaper;
    MoveL Offs(pOrigin,150.12,144.40,0.00),v40,fine,tPen\WObj:=wPaper;
    MoveL Offs(pOrigin,150.12,144.40,6.00),v60,z5,tPen\WObj:=wPaper;
    MoveL Offs(pOrigin,148.85,143.34,6.00),vTravel,z5,tPen\WObj:=wPaper;
    MoveL Offs(pOrigin,148.85,143.34,0.00),v60,z0,tPen\WObj:=wPaper;
    MoveL Offs(pOrigin,148.64,143.76,0.00),v40,z0,tPen\WObj:=wPaper;
    MoveL Offs(pOrigin,148.85,143.34,0.00),v40,fine,tPen\WObj:=wPaper;
    MoveL Offs(pOrigin,148.85,143.34,6.00),v60,z5,tPen\WObj:=wPaper;
    MoveL Offs(pOrigin,148.00,144.40,6.00),vTravel,z5,tPen\WObj:=wPaper;
    MoveL Offs(pOrigin,148.00,144.40,0.00),v60,z0,tPen\WObj:=wPaper;
    MoveL Offs(pOrigin,147.79,144.82,0.00),v40,z0,tPen\WObj:=wPaper;
    MoveL Offs(pOrigin,148.00,144.40,0.00),v40,z0,tPen\WObj:=wPaper;
    MoveL Offs(pOrigin,147.36,145.04,0.00),v40,z0,tPen\WObj:=wPaper;
    MoveL Offs(pOrigin,147.15,145.46,0.00),v40,z0,tPen\WObj:=wPaper;
    MoveL Offs(pOrigin,147.36,145.04,0.00),v40,fine,tPen\WObj:=wPaper;
    MoveL Offs(pOrigin,147.36,145.04,6.00),v60,z5,tPen\WObj:=wPaper;
    MoveL Offs(pOrigin,148.85,145.89,6.00),vTravel,z5,tPen\WObj:=wPaper;
    MoveL Offs(pOrigin,148.85,145.89,0.00),v60,z0,tPen\WObj:=wPaper;
    MoveL Offs(pOrigin,149.06,145.46,0.00),v40,z0,tPen\WObj:=wPaper;
    MoveL Offs(pOrigin,148.85,145.89,0.00),v40,fine,tPen\WObj:=wPaper;
    MoveL Offs(pOrigin,148.85,145.89,6.00),v60,z5,tPen\WObj:=wPaper;
    MoveL Offs(pOrigin,147.37,147.66,6.00),vTravel,z5,tPen\WObj:=wPaper;
    MoveL Offs(pOrigin,147.37,147.66,0.00),v60,z0,tPen\WObj:=wPaper;
    MoveL Offs(pOrigin,145.86,146.16,0.00),v40,z0,tPen\WObj:=wPaper;
    MoveL Offs(pOrigin,145.88,146.74,0.00),v40,z0,tPen\WObj:=wPaper;
    MoveL Offs(pOrigin,146.09,146.31,0.00),v40,z0,tPen\WObj:=wPaper;
    MoveL Offs(pOrigin,145.88,146.74,0.00),v40,z0,tPen\WObj:=wPaper;
    MoveL Offs(pOrigin,145.24,147.38,0.00),v40,z0,tPen\WObj:=wPaper;
    MoveL Offs(pOrigin,145.45,146.95,0.00),v40,z0,tPen\WObj:=wPaper;
    MoveL Offs(pOrigin,145.24,147.38,0.00),v40,z0,tPen\WObj:=wPaper;
    MoveL Offs(pOrigin,144.60,148.01,0.00),v40,z0,tPen\WObj:=wPaper;
    MoveL Offs(pOrigin,144.81,147.59,0.00),v40,z0,tPen\WObj:=wPaper;
    MoveL Offs(pOrigin,144.60,148.01,0.00),v40,z0,tPen\WObj:=wPaper;
    MoveL Offs(pOrigin,144.37,147.65,0.00),v40,z0,tPen\WObj:=wPaper;
    MoveL Offs(pOrigin,146.02,149.30,0.00),v40,fine,tPen\WObj:=wPaper;
    MoveL Offs(pOrigin,146.02,149.30,6.00),v60,z5,tPen\WObj:=wPaper;
    MoveL Offs(pOrigin,144.60,149.93,6.00),vTravel,z5,tPen\WObj:=wPaper;
    MoveL Offs(pOrigin,144.60,149.93,0.00),v60,z0,tPen\WObj:=wPaper;
    MoveL Offs(pOrigin,144.81,149.50,0.00),v40,z0,tPen\WObj:=wPaper;
    MoveL Offs(pOrigin,144.60,149.93,0.00),v40,z0,tPen\WObj:=wPaper;
    MoveL Offs(pOrigin,143.75,150.17,0.00),v40,z0,tPen\WObj:=wPaper;
    MoveL Offs(pOrigin,142.26,150.17,0.00),v40,z0,tPen\WObj:=wPaper;
    MoveL Offs(pOrigin,142.13,149.89,0.00),v40,z0,tPen\WObj:=wPaper;
    MoveL Offs(pOrigin,143.48,151.24,0.00),v40,z0,tPen\WObj:=wPaper;
    MoveL Offs(pOrigin,142.74,151.99,0.00),v40,z0,tPen\WObj:=wPaper;
    MoveL Offs(pOrigin,141.23,150.49,0.00),v40,z0,tPen\WObj:=wPaper;
    MoveL Offs(pOrigin,141.84,150.56,0.00),v40,z0,tPen\WObj:=wPaper;
    MoveL Offs(pOrigin,142.05,150.14,0.00),v40,z0,tPen\WObj:=wPaper;
    MoveL Offs(pOrigin,141.84,150.56,0.00),v40,z0,tPen\WObj:=wPaper;
    MoveL Offs(pOrigin,142.48,149.93,0.00),v40,z0,tPen\WObj:=wPaper;
    MoveL Offs(pOrigin,142.90,149.50,0.00),v40,z0,tPen\WObj:=wPaper;
    MoveL Offs(pOrigin,142.48,149.93,0.00),v40,fine,tPen\WObj:=wPaper;
    MoveL Offs(pOrigin,142.48,149.93,6.00),v60,z5,tPen\WObj:=wPaper;
    MoveL Offs(pOrigin,145.44,153.20,6.00),vTravel,z5,tPen\WObj:=wPaper;
    MoveL Offs(pOrigin,145.44,153.20,0.00),v60,z0,tPen\WObj:=wPaper;
    MoveL Offs(pOrigin,146.64,154.40,0.00),v40,z0,tPen\WObj:=wPaper;
    MoveL Offs(pOrigin,146.73,154.18,0.00),v40,z0,tPen\WObj:=wPaper;
    MoveL Offs(pOrigin,146.94,153.75,0.00),v40,z0,tPen\WObj:=wPaper;
    MoveL Offs(pOrigin,146.73,154.18,0.00),v40,z0,tPen\WObj:=wPaper;
    MoveL Offs(pOrigin,146.30,154.39,0.00),v40,z0,tPen\WObj:=wPaper;
    MoveL Offs(pOrigin,146.09,154.81,0.00),v40,z0,tPen\WObj:=wPaper;
    MoveL Offs(pOrigin,146.30,154.39,0.00),v40,z0,tPen\WObj:=wPaper;
    MoveL Offs(pOrigin,145.66,153.75,0.00),v40,z0,tPen\WObj:=wPaper;
    MoveL Offs(pOrigin,145.88,153.32,0.00),v40,z0,tPen\WObj:=wPaper;
    MoveL Offs(pOrigin,145.66,153.75,0.00),v40,z0,tPen\WObj:=wPaper;
    MoveL Offs(pOrigin,144.84,154.09,0.00),v40,z0,tPen\WObj:=wPaper;
    MoveL Offs(pOrigin,146.04,155.29,0.00),v40,z0,tPen\WObj:=wPaper;
    MoveL Offs(pOrigin,145.66,155.02,0.00),v40,z0,tPen\WObj:=wPaper;
    MoveL Offs(pOrigin,145.45,155.45,0.00),v40,z0,tPen\WObj:=wPaper;
    MoveL Offs(pOrigin,145.66,155.02,0.00),v40,z0,tPen\WObj:=wPaper;
    MoveL Offs(pOrigin,145.02,155.45,0.00),v40,z0,tPen\WObj:=wPaper;
    MoveL Offs(pOrigin,143.96,155.45,0.00),v40,z0,tPen\WObj:=wPaper;
    MoveL Offs(pOrigin,143.75,155.24,0.00),v40,z0,tPen\WObj:=wPaper;
    MoveL Offs(pOrigin,143.54,155.66,0.00),v40,z0,tPen\WObj:=wPaper;
    MoveL Offs(pOrigin,143.75,155.24,0.00),v40,z0,tPen\WObj:=wPaper;
    MoveL Offs(pOrigin,144.18,155.02,0.00),v40,z0,tPen\WObj:=wPaper;
    MoveL Offs(pOrigin,144.39,154.60,0.00),v40,z0,tPen\WObj:=wPaper;
    MoveL Offs(pOrigin,144.18,155.02,0.00),v40,z0,tPen\WObj:=wPaper;
    MoveL Offs(pOrigin,143.94,154.69,0.00),v40,z0,tPen\WObj:=wPaper;
    MoveL Offs(pOrigin,145.29,156.04,0.00),v40,z0,tPen\WObj:=wPaper;
    MoveL Offs(pOrigin,145.02,155.66,0.00),v40,z0,tPen\WObj:=wPaper;
    MoveL Offs(pOrigin,144.81,156.09,0.00),v40,z0,tPen\WObj:=wPaper;
    MoveL Offs(pOrigin,145.02,155.66,0.00),v40,fine,tPen\WObj:=wPaper;
    MoveL Offs(pOrigin,145.02,155.66,6.00),v60,z5,tPen\WObj:=wPaper;
    MoveL Offs(pOrigin,144.55,156.79,6.00),vTravel,z5,tPen\WObj:=wPaper;
    MoveL Offs(pOrigin,144.55,156.79,0.00),v60,z0,tPen\WObj:=wPaper;
    MoveL Offs(pOrigin,143.20,155.44,0.00),v40,z0,tPen\WObj:=wPaper;
    MoveL Offs(pOrigin,143.11,155.88,0.00),v40,z0,tPen\WObj:=wPaper;
    MoveL Offs(pOrigin,142.90,156.30,0.00),v40,z0,tPen\WObj:=wPaper;
    MoveL Offs(pOrigin,143.11,155.88,0.00),v40,z0,tPen\WObj:=wPaper;
    MoveL Offs(pOrigin,142.90,156.50,0.00),v40,z0,tPen\WObj:=wPaper;
    MoveL Offs(pOrigin,143.96,156.50,0.00),v40,z0,tPen\WObj:=wPaper;
    MoveL Offs(pOrigin,143.96,156.94,0.00),v40,z0,tPen\WObj:=wPaper;
    MoveL Offs(pOrigin,143.75,157.36,0.00),v40,z0,tPen\WObj:=wPaper;
    MoveL Offs(pOrigin,143.96,156.94,0.00),v40,z0,tPen\WObj:=wPaper;
    MoveL Offs(pOrigin,143.80,157.53,0.00),v40,z0,tPen\WObj:=wPaper;
    MoveL Offs(pOrigin,142.45,156.18,0.00),v40,z0,tPen\WObj:=wPaper;
    MoveL Offs(pOrigin,142.26,156.94,0.00),v40,z0,tPen\WObj:=wPaper;
    MoveL Offs(pOrigin,142.48,156.51,0.00),v40,z0,tPen\WObj:=wPaper;
    MoveL Offs(pOrigin,142.26,156.94,0.00),v40,z0,tPen\WObj:=wPaper;
    MoveL Offs(pOrigin,141.70,156.93,0.00),v40,z0,tPen\WObj:=wPaper;
  ENDPROC

  PROC DrawPart270()
    MoveL Offs(pOrigin,143.05,158.28,0.00),v40,z0,tPen\WObj:=wPaper;
    MoveL Offs(pOrigin,142.69,158.21,0.00),v40,z0,tPen\WObj:=wPaper;
    MoveL Offs(pOrigin,142.48,158.64,0.00),v40,z0,tPen\WObj:=wPaper;
    MoveL Offs(pOrigin,142.69,158.21,0.00),v40,z0,tPen\WObj:=wPaper;
    MoveL Offs(pOrigin,142.26,158.62,0.00),v40,z0,tPen\WObj:=wPaper;
    MoveL Offs(pOrigin,140.78,158.62,0.00),v40,z0,tPen\WObj:=wPaper;
    MoveL Offs(pOrigin,140.99,158.21,0.00),v40,z0,tPen\WObj:=wPaper;
    MoveL Offs(pOrigin,141.20,157.79,0.00),v40,z0,tPen\WObj:=wPaper;
    MoveL Offs(pOrigin,140.99,158.21,0.00),v40,z0,tPen\WObj:=wPaper;
    MoveL Offs(pOrigin,140.96,157.68,0.00),v40,z0,tPen\WObj:=wPaper;
    MoveL Offs(pOrigin,142.46,159.18,0.00),v40,z0,tPen\WObj:=wPaper;
    MoveL Offs(pOrigin,141.84,159.27,0.00),v40,z0,tPen\WObj:=wPaper;
    MoveL Offs(pOrigin,141.62,159.70,0.00),v40,z0,tPen\WObj:=wPaper;
    MoveL Offs(pOrigin,141.84,159.27,0.00),v40,z0,tPen\WObj:=wPaper;
    MoveL Offs(pOrigin,141.71,159.93,0.00),v40,z0,tPen\WObj:=wPaper;
    MoveL Offs(pOrigin,140.21,158.42,0.00),v40,z0,tPen\WObj:=wPaper;
    MoveL Offs(pOrigin,139.61,159.32,0.00),v40,z0,tPen\WObj:=wPaper;
    MoveL Offs(pOrigin,140.96,160.67,0.00),v40,z0,tPen\WObj:=wPaper;
    MoveL Offs(pOrigin,140.56,160.76,0.00),v40,z0,tPen\WObj:=wPaper;
    MoveL Offs(pOrigin,140.35,161.19,0.00),v40,z0,tPen\WObj:=wPaper;
    MoveL Offs(pOrigin,140.56,160.76,0.00),v40,z0,tPen\WObj:=wPaper;
    MoveL Offs(pOrigin,140.35,160.73,0.00),v40,z0,tPen\WObj:=wPaper;
    MoveL Offs(pOrigin,139.07,160.73,0.00),v40,z0,tPen\WObj:=wPaper;
    MoveL Offs(pOrigin,138.65,160.98,0.00),v40,z0,tPen\WObj:=wPaper;
    MoveL Offs(pOrigin,138.86,160.55,0.00),v40,z0,tPen\WObj:=wPaper;
    MoveL Offs(pOrigin,138.65,160.98,0.00),v40,z0,tPen\WObj:=wPaper;
    MoveL Offs(pOrigin,138.27,160.96,0.00),v40,z0,tPen\WObj:=wPaper;
    MoveL Offs(pOrigin,139.62,162.32,0.00),v40,z0,tPen\WObj:=wPaper;
    MoveL Offs(pOrigin,139.50,161.78,0.00),v40,z0,tPen\WObj:=wPaper;
    MoveL Offs(pOrigin,138.22,161.78,0.00),v40,z0,tPen\WObj:=wPaper;
    MoveL Offs(pOrigin,138.01,161.82,0.00),v40,z0,tPen\WObj:=wPaper;
    MoveL Offs(pOrigin,138.23,161.40,0.00),v40,z0,tPen\WObj:=wPaper;
    MoveL Offs(pOrigin,138.01,161.82,0.00),v40,z0,tPen\WObj:=wPaper;
    MoveL Offs(pOrigin,137.67,161.86,0.00),v40,z0,tPen\WObj:=wPaper;
    MoveL Offs(pOrigin,139.02,163.21,0.00),v40,z0,tPen\WObj:=wPaper;
    MoveL Offs(pOrigin,138.65,162.84,0.00),v40,z0,tPen\WObj:=wPaper;
    MoveL Offs(pOrigin,137.59,162.84,0.00),v40,z0,tPen\WObj:=wPaper;
    MoveL Offs(pOrigin,137.08,162.76,0.00),v40,z0,tPen\WObj:=wPaper;
    MoveL Offs(pOrigin,138.43,164.11,0.00),v40,z0,tPen\WObj:=wPaper;
    MoveL Offs(pOrigin,138.01,163.90,0.00),v40,z0,tPen\WObj:=wPaper;
    MoveL Offs(pOrigin,136.95,163.90,0.00),v40,z0,tPen\WObj:=wPaper;
    MoveL Offs(pOrigin,136.48,163.65,0.00),v40,z0,tPen\WObj:=wPaper;
    MoveL Offs(pOrigin,137.98,165.16,0.00),v40,z0,tPen\WObj:=wPaper;
    MoveL Offs(pOrigin,137.80,164.59,0.00),v40,z0,tPen\WObj:=wPaper;
    MoveL Offs(pOrigin,137.59,165.01,0.00),v40,z0,tPen\WObj:=wPaper;
    MoveL Offs(pOrigin,137.80,164.59,0.00),v40,z0,tPen\WObj:=wPaper;
    MoveL Offs(pOrigin,137.38,164.95,0.00),v40,z0,tPen\WObj:=wPaper;
    MoveL Offs(pOrigin,136.31,164.95,0.00),v40,z0,tPen\WObj:=wPaper;
    MoveL Offs(pOrigin,136.10,164.59,0.00),v40,z0,tPen\WObj:=wPaper;
    MoveL Offs(pOrigin,135.89,165.01,0.00),v40,z0,tPen\WObj:=wPaper;
    MoveL Offs(pOrigin,136.10,164.59,0.00),v40,z0,tPen\WObj:=wPaper;
    MoveL Offs(pOrigin,135.73,164.40,0.00),v40,z0,tPen\WObj:=wPaper;
    MoveL Offs(pOrigin,137.39,166.05,0.00),v40,z0,tPen\WObj:=wPaper;
    MoveL Offs(pOrigin,137.16,165.65,0.00),v40,z0,tPen\WObj:=wPaper;
    MoveL Offs(pOrigin,136.95,166.07,0.00),v40,z0,tPen\WObj:=wPaper;
    MoveL Offs(pOrigin,137.16,165.65,0.00),v40,z0,tPen\WObj:=wPaper;
    MoveL Offs(pOrigin,136.74,166.01,0.00),v40,z0,tPen\WObj:=wPaper;
    MoveL Offs(pOrigin,133.55,166.01,0.00),v40,z0,tPen\WObj:=wPaper;
    MoveL Offs(pOrigin,132.89,166.04,0.00),v40,z0,tPen\WObj:=wPaper;
    MoveL Offs(pOrigin,136.95,170.10,0.00),v40,z0,tPen\WObj:=wPaper;
    MoveL Offs(pOrigin,136.52,170.23,0.00),v40,z0,tPen\WObj:=wPaper;
    MoveL Offs(pOrigin,135.25,170.23,0.00),v40,z0,tPen\WObj:=wPaper;
    MoveL Offs(pOrigin,134.28,170.62,0.00),v40,z0,tPen\WObj:=wPaper;
    MoveL Offs(pOrigin,137.44,167.47,0.00),v40,z0,tPen\WObj:=wPaper;
    MoveL Offs(pOrigin,136.94,167.10,0.00),v40,z0,tPen\WObj:=wPaper;
    MoveL Offs(pOrigin,132.58,162.74,0.00),v40,fine,tPen\WObj:=wPaper;
    MoveL Offs(pOrigin,132.58,162.74,6.00),v60,z5,tPen\WObj:=wPaper;
    MoveL Offs(pOrigin,133.12,163.90,6.00),vTravel,z5,tPen\WObj:=wPaper;
    MoveL Offs(pOrigin,133.12,163.90,0.00),v60,z0,tPen\WObj:=wPaper;
    MoveL Offs(pOrigin,134.19,163.90,0.00),v40,fine,tPen\WObj:=wPaper;
    MoveL Offs(pOrigin,134.19,163.90,6.00),v60,z5,tPen\WObj:=wPaper;
    MoveL Offs(pOrigin,135.21,162.23,6.00),vTravel,z5,tPen\WObj:=wPaper;
    MoveL Offs(pOrigin,135.21,162.23,0.00),v60,z0,tPen\WObj:=wPaper;
    MoveL Offs(pOrigin,132.05,165.39,0.00),v40,z0,tPen\WObj:=wPaper;
    MoveL Offs(pOrigin,132.65,166.28,0.00),v40,z0,tPen\WObj:=wPaper;
    MoveL Offs(pOrigin,148.42,150.51,0.00),v40,fine,tPen\WObj:=wPaper;
    MoveL Offs(pOrigin,148.42,150.51,6.00),v60,z5,tPen\WObj:=wPaper;
    MoveL Offs(pOrigin,149.91,150.35,6.00),vTravel,z5,tPen\WObj:=wPaper;
    MoveL Offs(pOrigin,149.91,150.35,0.00),v60,z0,tPen\WObj:=wPaper;
    MoveL Offs(pOrigin,148.00,152.26,0.00),v40,z0,tPen\WObj:=wPaper;
    MoveL Offs(pOrigin,147.38,152.15,0.00),v40,z0,tPen\WObj:=wPaper;
    MoveL Offs(pOrigin,148.13,152.90,0.00),v40,z0,tPen\WObj:=wPaper;
    MoveL Offs(pOrigin,148.72,153.20,0.00),v40,z0,tPen\WObj:=wPaper;
    MoveL Offs(pOrigin,133.54,168.38,0.00),v40,z0,tPen\WObj:=wPaper;
    MoveL Offs(pOrigin,132.94,167.48,0.00),v40,z0,tPen\WObj:=wPaper;
    MoveL Offs(pOrigin,149.92,150.50,0.00),v40,fine,tPen\WObj:=wPaper;
    MoveL Offs(pOrigin,149.92,150.50,6.00),v60,z5,tPen\WObj:=wPaper;
    MoveL Offs(pOrigin,150.66,152.75,6.00),vTravel,z5,tPen\WObj:=wPaper;
    MoveL Offs(pOrigin,150.66,152.75,0.00),v60,z0,tPen\WObj:=wPaper;
    MoveL Offs(pOrigin,155.62,147.79,0.00),v40,z0,tPen\WObj:=wPaper;
    MoveL Offs(pOrigin,155.01,147.83,0.00),v40,z0,tPen\WObj:=wPaper;
    MoveL Offs(pOrigin,153.50,146.33,0.00),v40,z0,tPen\WObj:=wPaper;
    MoveL Offs(pOrigin,153.74,147.00,0.00),v40,z0,tPen\WObj:=wPaper;
    MoveL Offs(pOrigin,154.80,147.00,0.00),v40,z0,tPen\WObj:=wPaper;
    MoveL Offs(pOrigin,155.45,146.79,0.00),v40,z0,tPen\WObj:=wPaper;
    MoveL Offs(pOrigin,153.95,145.28,0.00),v40,z0,tPen\WObj:=wPaper;
    MoveL Offs(pOrigin,154.38,144.89,0.00),v40,z0,tPen\WObj:=wPaper;
    MoveL Offs(pOrigin,155.44,144.89,0.00),v40,fine,tPen\WObj:=wPaper;
    MoveL Offs(pOrigin,155.44,144.89,6.00),v60,z5,tPen\WObj:=wPaper;
    MoveL Offs(pOrigin,153.39,144.05,6.00),vTravel,z5,tPen\WObj:=wPaper;
    MoveL Offs(pOrigin,153.39,144.05,0.00),v60,z0,tPen\WObj:=wPaper;
    MoveL Offs(pOrigin,158.35,139.09,0.00),v40,z0,tPen\WObj:=wPaper;
    MoveL Offs(pOrigin,157.97,138.85,0.00),v40,z0,tPen\WObj:=wPaper;
    MoveL Offs(pOrigin,154.22,135.10,0.00),v40,fine,tPen\WObj:=wPaper;
    MoveL Offs(pOrigin,154.22,135.10,6.00),v60,z5,tPen\WObj:=wPaper;
    MoveL Offs(pOrigin,154.16,136.32,6.00),vTravel,z5,tPen\WObj:=wPaper;
    MoveL Offs(pOrigin,154.16,136.32,0.00),v60,z0,tPen\WObj:=wPaper;
    MoveL Offs(pOrigin,153.74,136.75,0.00),v40,z0,tPen\WObj:=wPaper;
    MoveL Offs(pOrigin,154.16,136.32,0.00),v40,z0,tPen\WObj:=wPaper;
    MoveL Offs(pOrigin,154.19,136.96,0.00),v40,z0,tPen\WObj:=wPaper;
    MoveL Offs(pOrigin,154.19,138.45,0.00),v40,z0,tPen\WObj:=wPaper;
    MoveL Offs(pOrigin,155.01,138.66,0.00),v40,z0,tPen\WObj:=wPaper;
    MoveL Offs(pOrigin,155.23,138.24,0.00),v40,z0,tPen\WObj:=wPaper;
    MoveL Offs(pOrigin,155.01,138.66,0.00),v40,z0,tPen\WObj:=wPaper;
    MoveL Offs(pOrigin,154.38,139.30,0.00),v40,z0,tPen\WObj:=wPaper;
    MoveL Offs(pOrigin,154.16,139.73,0.00),v40,z0,tPen\WObj:=wPaper;
    MoveL Offs(pOrigin,154.38,139.30,0.00),v40,z0,tPen\WObj:=wPaper;
    MoveL Offs(pOrigin,153.95,139.61,0.00),v40,z0,tPen\WObj:=wPaper;
    MoveL Offs(pOrigin,152.04,139.61,0.00),v40,z0,tPen\WObj:=wPaper;
    MoveL Offs(pOrigin,152.04,139.94,0.00),v40,z0,tPen\WObj:=wPaper;
  ENDPROC

  PROC DrawPart271()
    MoveL Offs(pOrigin,152.25,139.51,0.00),v40,z0,tPen\WObj:=wPaper;
    MoveL Offs(pOrigin,152.04,139.94,0.00),v40,fine,tPen\WObj:=wPaper;
    MoveL Offs(pOrigin,152.04,139.94,6.00),v60,z5,tPen\WObj:=wPaper;
    MoveL Offs(pOrigin,152.46,138.55,6.00),vTravel,z5,tPen\WObj:=wPaper;
    MoveL Offs(pOrigin,152.46,138.55,0.00),v60,z0,tPen\WObj:=wPaper;
    MoveL Offs(pOrigin,157.56,138.55,0.00),v40,fine,tPen\WObj:=wPaper;
    MoveL Offs(pOrigin,157.56,138.55,6.00),v60,z5,tPen\WObj:=wPaper;
    MoveL Offs(pOrigin,158.04,140.89,6.00),vTravel,z5,tPen\WObj:=wPaper;
    MoveL Offs(pOrigin,158.04,140.89,0.00),v60,z0,tPen\WObj:=wPaper;
    MoveL Offs(pOrigin,152.78,146.15,0.00),v40,fine,tPen\WObj:=wPaper;
    MoveL Offs(pOrigin,152.78,146.15,6.00),v60,z5,tPen\WObj:=wPaper;
    MoveL Offs(pOrigin,153.06,147.38,6.00),vTravel,z5,tPen\WObj:=wPaper;
    MoveL Offs(pOrigin,153.06,147.38,0.00),v60,z0,tPen\WObj:=wPaper;
    MoveL Offs(pOrigin,154.86,149.18,0.00),v40,z0,tPen\WObj:=wPaper;
    MoveL Offs(pOrigin,154.16,149.11,0.00),v40,z0,tPen\WObj:=wPaper;
    MoveL Offs(pOrigin,153.10,149.11,0.00),v40,z0,tPen\WObj:=wPaper;
    MoveL Offs(pOrigin,152.76,148.57,0.00),v40,z0,tPen\WObj:=wPaper;
    MoveL Offs(pOrigin,154.41,150.23,0.00),v40,z0,tPen\WObj:=wPaper;
    MoveL Offs(pOrigin,153.74,150.17,0.00),v40,z0,tPen\WObj:=wPaper;
    MoveL Offs(pOrigin,152.68,150.17,0.00),v40,z0,tPen\WObj:=wPaper;
    MoveL Offs(pOrigin,152.47,149.77,0.00),v40,z0,tPen\WObj:=wPaper;
    MoveL Offs(pOrigin,153.97,151.27,0.00),v40,z0,tPen\WObj:=wPaper;
    MoveL Offs(pOrigin,154.41,151.99,0.00),v40,z0,tPen\WObj:=wPaper;
    MoveL Offs(pOrigin,148.55,157.85,0.00),v40,fine,tPen\WObj:=wPaper;
    MoveL Offs(pOrigin,148.55,157.85,6.00),v60,z5,tPen\WObj:=wPaper;
    MoveL Offs(pOrigin,148.45,159.20,6.00),vTravel,z5,tPen\WObj:=wPaper;
    MoveL Offs(pOrigin,148.45,159.20,0.00),v60,z0,tPen\WObj:=wPaper;
    MoveL Offs(pOrigin,150.70,161.45,0.00),v40,z0,tPen\WObj:=wPaper;
    MoveL Offs(pOrigin,150.12,161.78,0.00),v40,z0,tPen\WObj:=wPaper;
    MoveL Offs(pOrigin,148.43,161.78,0.00),v40,z0,tPen\WObj:=wPaper;
    MoveL Offs(pOrigin,147.71,161.44,0.00),v40,z0,tPen\WObj:=wPaper;
    MoveL Offs(pOrigin,150.11,163.85,0.00),v40,z0,tPen\WObj:=wPaper;
    MoveL Offs(pOrigin,149.49,163.90,0.00),v40,z0,tPen\WObj:=wPaper;
    MoveL Offs(pOrigin,148.43,163.90,0.00),v40,z0,tPen\WObj:=wPaper;
    MoveL Offs(pOrigin,148.43,162.84,0.00),v40,z0,tPen\WObj:=wPaper;
    MoveL Offs(pOrigin,149.70,162.84,0.00),v40,fine,tPen\WObj:=wPaper;
    MoveL Offs(pOrigin,149.70,162.84,6.00),v60,z5,tPen\WObj:=wPaper;
    MoveL Offs(pOrigin,150.33,165.03,6.00),vTravel,z5,tPen\WObj:=wPaper;
    MoveL Offs(pOrigin,150.33,165.03,0.00),v60,z0,tPen\WObj:=wPaper;
    MoveL Offs(pOrigin,145.52,169.84,0.00),v40,z0,tPen\WObj:=wPaper;
    MoveL Offs(pOrigin,146.24,170.43,0.00),v40,z0,tPen\WObj:=wPaper;
    MoveL Offs(pOrigin,147.74,171.93,0.00),v40,fine,tPen\WObj:=wPaper;
    MoveL Offs(pOrigin,147.74,171.93,6.00),v60,z5,tPen\WObj:=wPaper;
    MoveL Offs(pOrigin,145.50,172.67,6.00),vTravel,z5,tPen\WObj:=wPaper;
    MoveL Offs(pOrigin,145.50,172.67,0.00),v60,z0,tPen\WObj:=wPaper;
    MoveL Offs(pOrigin,147.15,174.32,0.00),v40,fine,tPen\WObj:=wPaper;
    MoveL Offs(pOrigin,147.15,174.32,6.00),v60,z5,tPen\WObj:=wPaper;
    MoveL Offs(pOrigin,144.76,176.41,6.00),vTravel,z5,tPen\WObj:=wPaper;
    MoveL Offs(pOrigin,144.76,176.41,0.00),v60,z0,tPen\WObj:=wPaper;
    MoveL Offs(pOrigin,146.26,177.92,0.00),v40,fine,tPen\WObj:=wPaper;
    MoveL Offs(pOrigin,146.26,177.92,6.00),v60,z5,tPen\WObj:=wPaper;
    MoveL Offs(pOrigin,144.18,181.80,6.00),vTravel,z5,tPen\WObj:=wPaper;
    MoveL Offs(pOrigin,144.18,181.80,0.00),v60,z0,tPen\WObj:=wPaper;
    MoveL Offs(pOrigin,145.38,183.01,0.00),v40,fine,tPen\WObj:=wPaper;
    MoveL Offs(pOrigin,145.38,183.01,6.00),v60,z5,tPen\WObj:=wPaper;
    MoveL Offs(pOrigin,150.55,190.30,6.00),vTravel,z5,tPen\WObj:=wPaper;
    MoveL Offs(pOrigin,150.55,190.30,0.00),v60,z0,tPen\WObj:=wPaper;
    MoveL Offs(pOrigin,153.52,190.30,0.00),v40,z0,tPen\WObj:=wPaper;
    MoveL Offs(pOrigin,153.95,191.35,0.00),v40,z0,tPen\WObj:=wPaper;
    MoveL Offs(pOrigin,157.14,191.35,0.00),v40,z0,tPen\WObj:=wPaper;
    MoveL Offs(pOrigin,157.83,190.98,0.00),v40,z0,tPen\WObj:=wPaper;
    MoveL Offs(pOrigin,161.74,194.89,0.00),v40,fine,tPen\WObj:=wPaper;
    MoveL Offs(pOrigin,161.74,194.89,6.00),v60,z5,tPen\WObj:=wPaper;
    MoveL Offs(pOrigin,163.42,195.25,6.00),vTravel,z5,tPen\WObj:=wPaper;
    MoveL Offs(pOrigin,163.42,195.25,0.00),v60,z0,tPen\WObj:=wPaper;
    MoveL Offs(pOrigin,167.32,191.34,0.00),v40,z0,tPen\WObj:=wPaper;
    MoveL Offs(pOrigin,168.37,191.79,0.00),v40,z0,tPen\WObj:=wPaper;
    MoveL Offs(pOrigin,164.61,195.55,0.00),v40,z0,tPen\WObj:=wPaper;
    MoveL Offs(pOrigin,165.36,196.29,0.00),v40,z0,tPen\WObj:=wPaper;
    MoveL Offs(pOrigin,169.72,191.94,0.00),v40,z0,tPen\WObj:=wPaper;
    MoveL Offs(pOrigin,170.77,192.38,0.00),v40,z0,tPen\WObj:=wPaper;
    MoveL Offs(pOrigin,165.36,197.79,0.00),v40,z0,tPen\WObj:=wPaper;
    MoveL Offs(pOrigin,165.94,197.60,0.00),v40,z0,tPen\WObj:=wPaper;
    MoveL Offs(pOrigin,167.60,199.25,0.00),v40,z0,tPen\WObj:=wPaper;
    MoveL Offs(pOrigin,167.34,198.74,0.00),v40,z0,tPen\WObj:=wPaper;
    MoveL Offs(pOrigin,166.28,198.74,0.00),v40,z0,tPen\WObj:=wPaper;
    MoveL Offs(pOrigin,165.80,198.95,0.00),v40,z0,tPen\WObj:=wPaper;
    MoveL Offs(pOrigin,167.30,200.45,0.00),v40,fine,tPen\WObj:=wPaper;
    MoveL Offs(pOrigin,167.30,200.45,6.00),v60,z5,tPen\WObj:=wPaper;
    MoveL Offs(pOrigin,168.20,199.43,6.00),vTravel,z5,tPen\WObj:=wPaper;
    MoveL Offs(pOrigin,168.20,199.43,0.00),v60,z0,tPen\WObj:=wPaper;
    MoveL Offs(pOrigin,164.29,203.34,0.00),v40,z0,tPen\WObj:=wPaper;
    MoveL Offs(pOrigin,164.77,203.89,0.00),v40,z0,tPen\WObj:=wPaper;
    MoveL Offs(pOrigin,166.42,205.54,0.00),v40,fine,tPen\WObj:=wPaper;
    MoveL Offs(pOrigin,166.42,205.54,6.00),v60,z5,tPen\WObj:=wPaper;
    MoveL Offs(pOrigin,168.03,205.57,6.00),vTravel,z5,tPen\WObj:=wPaper;
    MoveL Offs(pOrigin,168.03,205.57,0.00),v60,z0,tPen\WObj:=wPaper;
    MoveL Offs(pOrigin,172.39,201.22,0.00),v40,z0,tPen\WObj:=wPaper;
    MoveL Offs(pOrigin,171.95,200.61,0.00),v40,z0,tPen\WObj:=wPaper;
    MoveL Offs(pOrigin,170.44,199.11,0.00),v40,z0,tPen\WObj:=wPaper;
    MoveL Offs(pOrigin,170.74,199.80,0.00),v40,z0,tPen\WObj:=wPaper;
    MoveL Offs(pOrigin,171.80,199.80,0.00),v40,z0,tPen\WObj:=wPaper;
    MoveL Offs(pOrigin,172.39,199.57,0.00),v40,z0,tPen\WObj:=wPaper;
    MoveL Offs(pOrigin,166.08,193.26,0.00),v40,fine,tPen\WObj:=wPaper;
    MoveL Offs(pOrigin,166.08,193.26,6.00),v60,z5,tPen\WObj:=wPaper;
    MoveL Offs(pOrigin,167.92,194.97,6.00),vTravel,z5,tPen\WObj:=wPaper;
    MoveL Offs(pOrigin,167.92,194.97,0.00),v60,z0,tPen\WObj:=wPaper;
    MoveL Offs(pOrigin,167.92,196.25,0.00),v40,fine,tPen\WObj:=wPaper;
    MoveL Offs(pOrigin,167.92,196.25,6.00),v60,z5,tPen\WObj:=wPaper;
    MoveL Offs(pOrigin,167.55,197.69,6.00),vTravel,z5,tPen\WObj:=wPaper;
    MoveL Offs(pOrigin,167.55,197.69,0.00),v60,z0,tPen\WObj:=wPaper;
    MoveL Offs(pOrigin,166.49,197.69,0.00),v40,fine,tPen\WObj:=wPaper;
    MoveL Offs(pOrigin,166.49,197.69,6.00),v60,z5,tPen\WObj:=wPaper;
    MoveL Offs(pOrigin,167.89,198.05,6.00),vTravel,z5,tPen\WObj:=wPaper;
    MoveL Offs(pOrigin,167.89,198.05,0.00),v60,z0,tPen\WObj:=wPaper;
    MoveL Offs(pOrigin,161.88,192.04,0.00),v40,z0,tPen\WObj:=wPaper;
    MoveL Offs(pOrigin,161.18,192.41,0.00),v40,z0,tPen\WObj:=wPaper;
    MoveL Offs(pOrigin,157.78,192.41,0.00),v40,z0,tPen\WObj:=wPaper;
    MoveL Offs(pOrigin,157.73,193.47,0.00),v40,z0,tPen\WObj:=wPaper;
    MoveL Offs(pOrigin,161.19,190.02,0.00),v40,fine,tPen\WObj:=wPaper;
    MoveL Offs(pOrigin,161.19,190.02,6.00),v60,z5,tPen\WObj:=wPaper;
    MoveL Offs(pOrigin,157.89,190.32,6.00),vTravel,z5,tPen\WObj:=wPaper;
    MoveL Offs(pOrigin,157.89,190.32,0.00),v60,z0,tPen\WObj:=wPaper;
    MoveL Offs(pOrigin,155.33,192.88,0.00),v40,fine,tPen\WObj:=wPaper;
    MoveL Offs(pOrigin,155.33,192.88,6.00),v60,z5,tPen\WObj:=wPaper;
    MoveL Offs(pOrigin,153.09,192.14,6.00),vTravel,z5,tPen\WObj:=wPaper;
    MoveL Offs(pOrigin,153.09,192.14,0.00),v60,z0,tPen\WObj:=wPaper;
    MoveL Offs(pOrigin,155.49,189.73,0.00),v40,fine,tPen\WObj:=wPaper;
    MoveL Offs(pOrigin,155.49,189.73,6.00),v60,z5,tPen\WObj:=wPaper;
    MoveL Offs(pOrigin,153.10,189.14,6.00),vTravel,z5,tPen\WObj:=wPaper;
  ENDPROC

  PROC DrawPart272()
    MoveL Offs(pOrigin,153.10,189.14,0.00),v60,z0,tPen\WObj:=wPaper;
    MoveL Offs(pOrigin,150.84,191.39,0.00),v40,fine,tPen\WObj:=wPaper;
    MoveL Offs(pOrigin,150.84,191.39,6.00),v60,z5,tPen\WObj:=wPaper;
    MoveL Offs(pOrigin,159.69,196.63,6.00),vTravel,z5,tPen\WObj:=wPaper;
    MoveL Offs(pOrigin,159.69,196.63,0.00),v60,z0,tPen\WObj:=wPaper;
    MoveL Offs(pOrigin,160.75,196.63,0.00),v40,fine,tPen\WObj:=wPaper;
    MoveL Offs(pOrigin,160.75,196.63,6.00),v60,z5,tPen\WObj:=wPaper;
    MoveL Offs(pOrigin,165.21,201.34,6.00),vTravel,z5,tPen\WObj:=wPaper;
    MoveL Offs(pOrigin,165.21,201.34,0.00),v60,z0,tPen\WObj:=wPaper;
    MoveL Offs(pOrigin,166.86,202.99,0.00),v40,z0,tPen\WObj:=wPaper;
    MoveL Offs(pOrigin,167.29,203.33,0.00),v40,z0,tPen\WObj:=wPaper;
    MoveL Offs(pOrigin,163.83,206.78,0.00),v40,z0,tPen\WObj:=wPaper;
    MoveL Offs(pOrigin,164.47,206.58,0.00),v40,z0,tPen\WObj:=wPaper;
    MoveL Offs(pOrigin,166.28,208.39,0.00),v40,z0,tPen\WObj:=wPaper;
    MoveL Offs(pOrigin,166.82,208.27,0.00),v40,z0,tPen\WObj:=wPaper;
    MoveL Offs(pOrigin,163.67,211.43,0.00),v40,fine,tPen\WObj:=wPaper;
    MoveL Offs(pOrigin,163.67,211.43,6.00),v60,z5,tPen\WObj:=wPaper;
    MoveL Offs(pOrigin,164.33,209.43,6.00),vTravel,z5,tPen\WObj:=wPaper;
    MoveL Offs(pOrigin,164.33,209.43,0.00),v60,z0,tPen\WObj:=wPaper;
    MoveL Offs(pOrigin,166.14,211.23,0.00),v40,fine,tPen\WObj:=wPaper;
    MoveL Offs(pOrigin,166.14,211.23,6.00),v60,z5,tPen\WObj:=wPaper;
    MoveL Offs(pOrigin,170.32,207.95,6.00),vTravel,z5,tPen\WObj:=wPaper;
    MoveL Offs(pOrigin,170.32,207.95,0.00),v60,z0,tPen\WObj:=wPaper;
    MoveL Offs(pOrigin,168.52,206.15,0.00),v40,fine,tPen\WObj:=wPaper;
    MoveL Offs(pOrigin,168.52,206.15,6.00),v60,z5,tPen\WObj:=wPaper;
    MoveL Offs(pOrigin,161.74,205.89,6.00),vTravel,z5,tPen\WObj:=wPaper;
    MoveL Offs(pOrigin,161.74,205.89,0.00),v60,z0,tPen\WObj:=wPaper;
    MoveL Offs(pOrigin,159.03,208.60,0.00),v40,fine,tPen\WObj:=wPaper;
    MoveL Offs(pOrigin,159.03,208.60,6.00),v60,z5,tPen\WObj:=wPaper;
    MoveL Offs(pOrigin,159.90,206.14,6.00),vTravel,z5,tPen\WObj:=wPaper;
    MoveL Offs(pOrigin,159.90,206.14,0.00),v60,z0,tPen\WObj:=wPaper;
    MoveL Offs(pOrigin,160.96,206.14,0.00),v40,fine,tPen\WObj:=wPaper;
    MoveL Offs(pOrigin,160.96,206.14,6.00),v60,z5,tPen\WObj:=wPaper;
    MoveL Offs(pOrigin,162.61,215.48,6.00),vTravel,z5,tPen\WObj:=wPaper;
    MoveL Offs(pOrigin,162.61,215.48,0.00),v60,z0,tPen\WObj:=wPaper;
    MoveL Offs(pOrigin,160.05,218.03,0.00),v40,fine,tPen\WObj:=wPaper;
    MoveL Offs(pOrigin,160.05,218.03,6.00),v60,z5,tPen\WObj:=wPaper;
    MoveL Offs(pOrigin,164.66,218.72,6.00),vTravel,z5,tPen\WObj:=wPaper;
    MoveL Offs(pOrigin,164.66,218.72,0.00),v60,z0,tPen\WObj:=wPaper;
    MoveL Offs(pOrigin,167.07,221.12,0.00),v40,fine,tPen\WObj:=wPaper;
    MoveL Offs(pOrigin,167.07,221.12,6.00),v60,z5,tPen\WObj:=wPaper;
    MoveL Offs(pOrigin,169.68,223.03,6.00),vTravel,z5,tPen\WObj:=wPaper;
    MoveL Offs(pOrigin,169.68,223.03,0.00),v60,z0,tPen\WObj:=wPaper;
    MoveL Offs(pOrigin,170.74,223.03,0.00),v40,z0,tPen\WObj:=wPaper;
    MoveL Offs(pOrigin,171.72,222.79,0.00),v40,z0,tPen\WObj:=wPaper;
    MoveL Offs(pOrigin,165.71,228.80,0.00),v40,z0,tPen\WObj:=wPaper;
    MoveL Offs(pOrigin,164.96,228.05,0.00),v40,z0,tPen\WObj:=wPaper;
    MoveL Offs(pOrigin,171.27,221.74,0.00),v40,fine,tPen\WObj:=wPaper;
    MoveL Offs(pOrigin,171.27,221.74,6.00),v60,z5,tPen\WObj:=wPaper;
    MoveL Offs(pOrigin,170.68,219.35,6.00),vTravel,z5,tPen\WObj:=wPaper;
    MoveL Offs(pOrigin,170.68,219.35,0.00),v60,z0,tPen\WObj:=wPaper;
    MoveL Offs(pOrigin,163.77,226.26,0.00),v40,fine,tPen\WObj:=wPaper;
    MoveL Offs(pOrigin,163.77,226.26,6.00),v60,z5,tPen\WObj:=wPaper;
    MoveL Offs(pOrigin,165.42,227.26,6.00),vTravel,z5,tPen\WObj:=wPaper;
    MoveL Offs(pOrigin,165.42,227.26,0.00),v60,z0,tPen\WObj:=wPaper;
    MoveL Offs(pOrigin,166.91,227.26,0.00),v40,z0,tPen\WObj:=wPaper;
    MoveL Offs(pOrigin,166.70,226.85,0.00),v40,z0,tPen\WObj:=wPaper;
    MoveL Offs(pOrigin,168.82,228.98,0.00),v40,z0,tPen\WObj:=wPaper;
    MoveL Offs(pOrigin,166.70,226.85,0.00),v40,fine,tPen\WObj:=wPaper;
    MoveL Offs(pOrigin,166.70,226.85,6.00),v60,z5,tPen\WObj:=wPaper;
    MoveL Offs(pOrigin,170.52,225.14,6.00),vTravel,z5,tPen\WObj:=wPaper;
    MoveL Offs(pOrigin,170.52,225.14,0.00),v60,z0,tPen\WObj:=wPaper;
    MoveL Offs(pOrigin,171.59,225.14,0.00),v40,z0,tPen\WObj:=wPaper;
    MoveL Offs(pOrigin,171.16,226.20,0.00),v40,z0,tPen\WObj:=wPaper;
    MoveL Offs(pOrigin,172.23,226.20,0.00),v40,fine,tPen\WObj:=wPaper;
    MoveL Offs(pOrigin,172.23,226.20,6.00),v60,z5,tPen\WObj:=wPaper;
    MoveL Offs(pOrigin,170.74,230.42,6.00),vTravel,z5,tPen\WObj:=wPaper;
    MoveL Offs(pOrigin,170.74,230.42,0.00),v60,z0,tPen\WObj:=wPaper;
    MoveL Offs(pOrigin,169.04,230.42,0.00),v40,fine,tPen\WObj:=wPaper;
    MoveL Offs(pOrigin,169.04,230.42,6.00),v60,z5,tPen\WObj:=wPaper;
    MoveL Offs(pOrigin,162.58,224.46,6.00),vTravel,z5,tPen\WObj:=wPaper;
    MoveL Offs(pOrigin,162.58,224.46,0.00),v60,z0,tPen\WObj:=wPaper;
    MoveL Offs(pOrigin,170.24,216.80,0.00),v40,fine,tPen\WObj:=wPaper;
    MoveL Offs(pOrigin,170.24,216.80,6.00),v60,z5,tPen\WObj:=wPaper;
    MoveL Offs(pOrigin,184.12,228.34,6.00),vTravel,z5,tPen\WObj:=wPaper;
    MoveL Offs(pOrigin,184.12,228.34,0.00),v60,z0,tPen\WObj:=wPaper;
    MoveL Offs(pOrigin,184.55,228.55,0.00),v40,z0,tPen\WObj:=wPaper;
    MoveL Offs(pOrigin,184.12,228.34,0.00),v40,fine,tPen\WObj:=wPaper;
    MoveL Offs(pOrigin,184.12,228.34,6.00),v60,z5,tPen\WObj:=wPaper;
    MoveL Offs(pOrigin,188.77,231.13,6.00),vTravel,z5,tPen\WObj:=wPaper;
    MoveL Offs(pOrigin,188.77,231.13,0.00),v60,z0,tPen\WObj:=wPaper;
    MoveL Offs(pOrigin,190.88,229.02,0.00),v40,z0,tPen\WObj:=wPaper;
    MoveL Offs(pOrigin,191.92,229.47,0.00),v40,z0,tPen\WObj:=wPaper;
    MoveL Offs(pOrigin,189.97,231.42,0.00),v40,fine,tPen\WObj:=wPaper;
    MoveL Offs(pOrigin,189.97,231.42,6.00),v60,z5,tPen\WObj:=wPaper;
    MoveL Offs(pOrigin,192.06,232.31,6.00),vTravel,z5,tPen\WObj:=wPaper;
    MoveL Offs(pOrigin,192.06,232.31,0.00),v60,z0,tPen\WObj:=wPaper;
    MoveL Offs(pOrigin,194.32,230.06,0.00),v40,fine,tPen\WObj:=wPaper;
    MoveL Offs(pOrigin,194.32,230.06,6.00),v60,z5,tPen\WObj:=wPaper;
    MoveL Offs(pOrigin,196.56,230.80,6.00),vTravel,z5,tPen\WObj:=wPaper;
    MoveL Offs(pOrigin,196.56,230.80,0.00),v60,z0,tPen\WObj:=wPaper;
    MoveL Offs(pOrigin,194.46,232.91,0.00),v40,fine,tPen\WObj:=wPaper;
    MoveL Offs(pOrigin,194.46,232.91,6.00),v60,z5,tPen\WObj:=wPaper;
    MoveL Offs(pOrigin,193.85,236.50,6.00),vTravel,z5,tPen\WObj:=wPaper;
    MoveL Offs(pOrigin,193.85,236.50,0.00),v60,z0,tPen\WObj:=wPaper;
    MoveL Offs(pOrigin,191.29,239.06,0.00),v40,fine,tPen\WObj:=wPaper;
    MoveL Offs(pOrigin,191.29,239.06,6.00),v60,z5,tPen\WObj:=wPaper;
    MoveL Offs(pOrigin,230.50,252.12,6.00),vTravel,z5,tPen\WObj:=wPaper;
    MoveL Offs(pOrigin,230.50,252.12,0.00),v60,z0,tPen\WObj:=wPaper;
    MoveL Offs(pOrigin,232.30,250.32,0.00),v40,z0,tPen\WObj:=wPaper;
    MoveL Offs(pOrigin,233.20,250.91,0.00),v40,z0,tPen\WObj:=wPaper;
    MoveL Offs(pOrigin,231.70,252.41,0.00),v40,z0,tPen\WObj:=wPaper;
    MoveL Offs(pOrigin,232.60,253.01,0.00),v40,z0,tPen\WObj:=wPaper;
    MoveL Offs(pOrigin,234.25,251.36,0.00),v40,fine,tPen\WObj:=wPaper;
    MoveL Offs(pOrigin,234.25,251.36,6.00),v60,z5,tPen\WObj:=wPaper;
    MoveL Offs(pOrigin,232.46,248.67,6.00),vTravel,z5,tPen\WObj:=wPaper;
    MoveL Offs(pOrigin,232.46,248.67,0.00),v60,z0,tPen\WObj:=wPaper;
    MoveL Offs(pOrigin,233.66,247.47,0.00),v40,fine,tPen\WObj:=wPaper;
    MoveL Offs(pOrigin,233.66,247.47,6.00),v60,z5,tPen\WObj:=wPaper;
    MoveL Offs(pOrigin,254.04,238.96,6.00),vTravel,z5,tPen\WObj:=wPaper;
    MoveL Offs(pOrigin,254.04,238.96,0.00),v60,z0,tPen\WObj:=wPaper;
    MoveL Offs(pOrigin,254.46,238.96,0.00),v40,z0,tPen\WObj:=wPaper;
    MoveL Offs(pOrigin,254.68,238.54,0.00),v40,fine,tPen\WObj:=wPaper;
    MoveL Offs(pOrigin,254.68,238.54,6.00),v60,z5,tPen\WObj:=wPaper;
    MoveL Offs(pOrigin,255.52,240.45,6.00),vTravel,z5,tPen\WObj:=wPaper;
    MoveL Offs(pOrigin,255.52,240.45,0.00),v60,z0,tPen\WObj:=wPaper;
    MoveL Offs(pOrigin,255.95,240.24,0.00),v40,z0,tPen\WObj:=wPaper;
    MoveL Offs(pOrigin,255.52,240.45,0.00),v40,fine,tPen\WObj:=wPaper;
    MoveL Offs(pOrigin,255.52,240.45,6.00),v60,z5,tPen\WObj:=wPaper;
    MoveL Offs(pOrigin,259.23,232.64,6.00),vTravel,z5,tPen\WObj:=wPaper;
  ENDPROC

  PROC DrawPart273()
    MoveL Offs(pOrigin,259.23,232.64,0.00),v60,z0,tPen\WObj:=wPaper;
    MoveL Offs(pOrigin,267.79,241.20,0.00),v40,fine,tPen\WObj:=wPaper;
    MoveL Offs(pOrigin,267.79,241.20,6.00),v60,z5,tPen\WObj:=wPaper;
    MoveL Offs(pOrigin,251.85,227.79,6.00),vTravel,z5,tPen\WObj:=wPaper;
    MoveL Offs(pOrigin,251.85,227.79,0.00),v60,z0,tPen\WObj:=wPaper;
    MoveL Offs(pOrigin,251.10,228.54,0.00),v40,z0,tPen\WObj:=wPaper;
    MoveL Offs(pOrigin,250.50,227.64,0.00),v40,z0,tPen\WObj:=wPaper;
    MoveL Offs(pOrigin,249.60,228.54,0.00),v40,fine,tPen\WObj:=wPaper;
    MoveL Offs(pOrigin,249.60,228.54,6.00),v60,z5,tPen\WObj:=wPaper;
    MoveL Offs(pOrigin,248.40,228.25,6.00),vTravel,z5,tPen\WObj:=wPaper;
    MoveL Offs(pOrigin,248.40,228.25,0.00),v60,z0,tPen\WObj:=wPaper;
    MoveL Offs(pOrigin,249.45,227.19,0.00),v40,z0,tPen\WObj:=wPaper;
    MoveL Offs(pOrigin,248.41,226.75,0.00),v40,z0,tPen\WObj:=wPaper;
    MoveL Offs(pOrigin,247.05,228.10,0.00),v40,fine,tPen\WObj:=wPaper;
    MoveL Offs(pOrigin,247.05,228.10,6.00),v60,z5,tPen\WObj:=wPaper;
    MoveL Offs(pOrigin,245.86,227.80,6.00),vTravel,z5,tPen\WObj:=wPaper;
    MoveL Offs(pOrigin,245.86,227.80,0.00),v60,z0,tPen\WObj:=wPaper;
    MoveL Offs(pOrigin,248.56,225.10,0.00),v40,fine,tPen\WObj:=wPaper;
    MoveL Offs(pOrigin,248.56,225.10,6.00),v60,z5,tPen\WObj:=wPaper;
    MoveL Offs(pOrigin,250.64,225.36,6.00),vTravel,z5,tPen\WObj:=wPaper;
    MoveL Offs(pOrigin,250.64,225.36,0.00),v60,z0,tPen\WObj:=wPaper;
    MoveL Offs(pOrigin,245.54,225.15,0.00),v40,z0,tPen\WObj:=wPaper;
    MoveL Offs(pOrigin,242.56,224.30,0.00),v40,fine,tPen\WObj:=wPaper;
    MoveL Offs(pOrigin,242.56,224.30,6.00),v60,z5,tPen\WObj:=wPaper;
    MoveL Offs(pOrigin,243.77,225.41,6.00),vTravel,z5,tPen\WObj:=wPaper;
    MoveL Offs(pOrigin,243.77,225.41,0.00),v60,z0,tPen\WObj:=wPaper;
    MoveL Offs(pOrigin,244.97,224.21,0.00),v40,fine,tPen\WObj:=wPaper;
    MoveL Offs(pOrigin,244.97,224.21,6.00),v60,z5,tPen\WObj:=wPaper;
    MoveL Offs(pOrigin,289.86,239.05,6.00),vTravel,z5,tPen\WObj:=wPaper;
    MoveL Offs(pOrigin,289.86,239.05,0.00),v60,z0,tPen\WObj:=wPaper;
    MoveL Offs(pOrigin,292.57,236.35,0.00),v40,fine,tPen\WObj:=wPaper;
    MoveL Offs(pOrigin,292.57,236.35,6.00),v60,z5,tPen\WObj:=wPaper;
    MoveL Offs(pOrigin,295.55,240.83,6.00),vTravel,z5,tPen\WObj:=wPaper;
    MoveL Offs(pOrigin,295.55,240.83,0.00),v60,z0,tPen\WObj:=wPaper;
    MoveL Offs(pOrigin,297.95,238.43,0.00),v40,fine,tPen\WObj:=wPaper;
    MoveL Offs(pOrigin,297.95,238.43,6.00),v60,z5,tPen\WObj:=wPaper;
    MoveL Offs(pOrigin,290.76,258.20,6.00),vTravel,z5,tPen\WObj:=wPaper;
    MoveL Offs(pOrigin,290.76,258.20,0.00),v60,z0,tPen\WObj:=wPaper;
    MoveL Offs(pOrigin,291.82,259.25,0.00),v40,fine,tPen\WObj:=wPaper;
    MoveL Offs(pOrigin,291.82,259.25,6.00),v60,z5,tPen\WObj:=wPaper;
    MoveL Offs(pOrigin,293.56,269.77,6.00),vTravel,z5,tPen\WObj:=wPaper;
    MoveL Offs(pOrigin,293.56,269.77,0.00),v60,z0,tPen\WObj:=wPaper;
    MoveL Offs(pOrigin,294.20,270.41,0.00),v40,z0,tPen\WObj:=wPaper;
    MoveL Offs(pOrigin,293.56,269.77,0.00),v40,fine,tPen\WObj:=wPaper;
    MoveL Offs(pOrigin,293.56,269.77,6.00),v60,z5,tPen\WObj:=wPaper;
    MoveL Offs(pOrigin,295.75,271.99,6.00),vTravel,z5,tPen\WObj:=wPaper;
    MoveL Offs(pOrigin,295.75,271.99,0.00),v60,z0,tPen\WObj:=wPaper;
    MoveL Offs(pOrigin,303.87,263.88,0.00),v40,fine,tPen\WObj:=wPaper;
    MoveL Offs(pOrigin,303.87,263.88,6.00),v60,z5,tPen\WObj:=wPaper;
    MoveL Offs(pOrigin,301.42,265.87,6.00),vTravel,z5,tPen\WObj:=wPaper;
    MoveL Offs(pOrigin,301.42,265.87,0.00),v60,z0,tPen\WObj:=wPaper;
    MoveL Offs(pOrigin,303.08,267.53,0.00),v40,fine,tPen\WObj:=wPaper;
    MoveL Offs(pOrigin,303.08,267.53,6.00),v60,z5,tPen\WObj:=wPaper;
    MoveL Offs(pOrigin,227.05,269.77,6.00),vTravel,z5,tPen\WObj:=wPaper;
    MoveL Offs(pOrigin,227.05,269.77,0.00),v60,z0,tPen\WObj:=wPaper;
    MoveL Offs(pOrigin,227.05,271.05,0.00),v40,z0,tPen\WObj:=wPaper;
    MoveL Offs(pOrigin,226.00,270.84,0.00),v40,z0,tPen\WObj:=wPaper;
    MoveL Offs(pOrigin,226.00,269.77,0.00),v40,z0,tPen\WObj:=wPaper;
    MoveL Offs(pOrigin,224.94,269.77,0.00),v40,z0,tPen\WObj:=wPaper;
    MoveL Offs(pOrigin,224.94,270.84,0.00),v40,fine,tPen\WObj:=wPaper;
    MoveL Offs(pOrigin,224.94,270.84,6.00),v60,z5,tPen\WObj:=wPaper;
    MoveL Offs(pOrigin,277.41,180.79,6.00),vTravel,z5,tPen\WObj:=wPaper;
    MoveL Offs(pOrigin,277.41,180.79,0.00),v60,z0,tPen\WObj:=wPaper;
    MoveL Offs(pOrigin,278.90,180.79,0.00),v40,z0,tPen\WObj:=wPaper;
    MoveL Offs(pOrigin,279.29,181.02,0.00),v40,z0,tPen\WObj:=wPaper;
    MoveL Offs(pOrigin,277.19,178.92,0.00),v40,fine,tPen\WObj:=wPaper;
    MoveL Offs(pOrigin,277.19,178.92,6.00),v60,z5,tPen\WObj:=wPaper;
    MoveL Offs(pOrigin,306.27,185.60,6.00),vTravel,z5,tPen\WObj:=wPaper;
    MoveL Offs(pOrigin,306.27,185.60,0.00),v60,z0,tPen\WObj:=wPaper;
    MoveL Offs(pOrigin,307.62,186.95,0.00),v40,fine,tPen\WObj:=wPaper;
    MoveL Offs(pOrigin,307.62,186.95,6.00),v60,z5,tPen\WObj:=wPaper;
    MoveL Offs(pOrigin,357.22,156.76,6.00),vTravel,z5,tPen\WObj:=wPaper;
    MoveL Offs(pOrigin,357.22,156.76,0.00),v60,z0,tPen\WObj:=wPaper;
    MoveL Offs(pOrigin,359.78,154.20,0.00),v40,z0,tPen\WObj:=wPaper;
    MoveL Offs(pOrigin,359.01,154.39,0.00),v40,z0,tPen\WObj:=wPaper;
    MoveL Offs(pOrigin,357.95,154.39,0.00),v40,z0,tPen\WObj:=wPaper;
    MoveL Offs(pOrigin,357.52,153.34,0.00),v40,z0,tPen\WObj:=wPaper;
    MoveL Offs(pOrigin,358.59,153.34,0.00),v40,fine,tPen\WObj:=wPaper;
    MoveL Offs(pOrigin,358.59,153.34,6.00),v60,z5,tPen\WObj:=wPaper;
    MoveL Offs(pOrigin,356.34,153.16,6.00),vTravel,z5,tPen\WObj:=wPaper;
    MoveL Offs(pOrigin,356.34,153.16,0.00),v60,z0,tPen\WObj:=wPaper;
    MoveL Offs(pOrigin,359.04,150.46,0.00),v40,fine,tPen\WObj:=wPaper;
    MoveL Offs(pOrigin,359.04,150.46,6.00),v60,z5,tPen\WObj:=wPaper;
    MoveL Offs(pOrigin,358.30,148.22,6.00),vTravel,z5,tPen\WObj:=wPaper;
    MoveL Offs(pOrigin,358.30,148.22,0.00),v60,z0,tPen\WObj:=wPaper;
    MoveL Offs(pOrigin,355.74,150.77,0.00),v40,fine,tPen\WObj:=wPaper;
    MoveL Offs(pOrigin,355.74,150.77,6.00),v60,z5,tPen\WObj:=wPaper;
    MoveL Offs(pOrigin,355.15,148.37,6.00),vTravel,z5,tPen\WObj:=wPaper;
    MoveL Offs(pOrigin,355.15,148.37,0.00),v60,z0,tPen\WObj:=wPaper;
    MoveL Offs(pOrigin,357.71,145.82,0.00),v40,fine,tPen\WObj:=wPaper;
    MoveL Offs(pOrigin,357.71,145.82,6.00),v60,z5,tPen\WObj:=wPaper;
    MoveL Offs(pOrigin,356.67,144.89,6.00),vTravel,z5,tPen\WObj:=wPaper;
    MoveL Offs(pOrigin,356.67,144.89,0.00),v60,z0,tPen\WObj:=wPaper;
    MoveL Offs(pOrigin,355.40,144.89,0.00),v40,fine,tPen\WObj:=wPaper;
    MoveL Offs(pOrigin,355.40,144.89,6.00),v60,z5,tPen\WObj:=wPaper;
    MoveL Offs(pOrigin,360.26,143.27,6.00),vTravel,z5,tPen\WObj:=wPaper;
    MoveL Offs(pOrigin,360.26,143.27,0.00),v60,z0,tPen\WObj:=wPaper;
    MoveL Offs(pOrigin,366.27,137.26,0.00),v40,z0,tPen\WObj:=wPaper;
    MoveL Offs(pOrigin,365.53,136.51,0.00),v40,z0,tPen\WObj:=wPaper;
    MoveL Offs(pOrigin,359.82,142.22,0.00),v40,fine,tPen\WObj:=wPaper;
    MoveL Offs(pOrigin,359.82,142.22,6.00),v60,z5,tPen\WObj:=wPaper;
    MoveL Offs(pOrigin,361.45,145.06,6.00),vTravel,z5,tPen\WObj:=wPaper;
    MoveL Offs(pOrigin,361.45,145.06,0.00),v60,z0,tPen\WObj:=wPaper;
    MoveL Offs(pOrigin,365.21,141.30,0.00),v40,z0,tPen\WObj:=wPaper;
    MoveL Offs(pOrigin,364.33,141.64,0.00),v40,z0,tPen\WObj:=wPaper;
    MoveL Offs(pOrigin,365.17,142.49,0.00),v40,z0,tPen\WObj:=wPaper;
    MoveL Offs(pOrigin,364.33,141.64,0.00),v40,fine,tPen\WObj:=wPaper;
    MoveL Offs(pOrigin,364.33,141.64,6.00),v60,z5,tPen\WObj:=wPaper;
    MoveL Offs(pOrigin,364.33,143.12,6.00),vTravel,z5,tPen\WObj:=wPaper;
    MoveL Offs(pOrigin,364.33,143.12,0.00),v60,z0,tPen\WObj:=wPaper;
    MoveL Offs(pOrigin,364.75,143.55,0.00),v40,z0,tPen\WObj:=wPaper;
    MoveL Offs(pOrigin,364.33,143.12,0.00),v40,fine,tPen\WObj:=wPaper;
    MoveL Offs(pOrigin,364.33,143.12,6.00),v60,z5,tPen\WObj:=wPaper;
    MoveL Offs(pOrigin,365.96,142.05,6.00),vTravel,z5,tPen\WObj:=wPaper;
    MoveL Offs(pOrigin,365.96,142.05,0.00),v60,z0,tPen\WObj:=wPaper;
    MoveL Offs(pOrigin,362.05,145.96,0.00),v40,fine,tPen\WObj:=wPaper;
    MoveL Offs(pOrigin,362.05,145.96,6.00),v60,z5,tPen\WObj:=wPaper;
    MoveL Offs(pOrigin,365.39,138.88,6.00),vTravel,z5,tPen\WObj:=wPaper;
    MoveL Offs(pOrigin,365.39,138.88,0.00),v60,z0,tPen\WObj:=wPaper;
    MoveL Offs(pOrigin,365.81,139.30,0.00),v40,z0,tPen\WObj:=wPaper;
  ENDPROC

  PROC DrawPart274()
    MoveL Offs(pOrigin,365.39,138.88,0.00),v40,z0,tPen\WObj:=wPaper;
    MoveL Offs(pOrigin,365.17,138.55,0.00),v40,z0,tPen\WObj:=wPaper;
    MoveL Offs(pOrigin,366.45,138.55,0.00),v40,z0,tPen\WObj:=wPaper;
    MoveL Offs(pOrigin,367.09,138.88,0.00),v40,z0,tPen\WObj:=wPaper;
    MoveL Offs(pOrigin,367.51,139.30,0.00),v40,z0,tPen\WObj:=wPaper;
    MoveL Offs(pOrigin,367.09,138.88,0.00),v40,fine,tPen\WObj:=wPaper;
    MoveL Offs(pOrigin,367.09,138.88,6.00),v60,z5,tPen\WObj:=wPaper;
    MoveL Offs(pOrigin,363.48,137.39,6.00),vTravel,z5,tPen\WObj:=wPaper;
    MoveL Offs(pOrigin,363.48,137.39,0.00),v60,z0,tPen\WObj:=wPaper;
    MoveL Offs(pOrigin,363.90,137.81,0.00),v40,z0,tPen\WObj:=wPaper;
    MoveL Offs(pOrigin,363.48,137.39,0.00),v40,fine,tPen\WObj:=wPaper;
    MoveL Offs(pOrigin,363.48,137.39,6.00),v60,z5,tPen\WObj:=wPaper;
    MoveL Offs(pOrigin,374.21,136.78,6.00),vTravel,z5,tPen\WObj:=wPaper;
    MoveL Offs(pOrigin,374.21,136.78,0.00),v60,z0,tPen\WObj:=wPaper;
    MoveL Offs(pOrigin,377.07,133.93,0.00),v40,fine,tPen\WObj:=wPaper;
    MoveL Offs(pOrigin,377.07,133.93,6.00),v60,z5,tPen\WObj:=wPaper;
    MoveL Offs(pOrigin,385.45,143.76,6.00),vTravel,z5,tPen\WObj:=wPaper;
    MoveL Offs(pOrigin,385.45,143.76,0.00),v60,z0,tPen\WObj:=wPaper;
    MoveL Offs(pOrigin,385.45,145.89,0.00),v40,fine,tPen\WObj:=wPaper;
    MoveL Offs(pOrigin,385.45,145.89,6.00),v60,z5,tPen\WObj:=wPaper;
    MoveL Offs(pOrigin,371.12,154.39,6.00),vTravel,z5,tPen\WObj:=wPaper;
    MoveL Offs(pOrigin,371.12,154.39,0.00),v60,z0,tPen\WObj:=wPaper;
    MoveL Offs(pOrigin,370.06,154.39,0.00),v40,fine,tPen\WObj:=wPaper;
    MoveL Offs(pOrigin,370.06,154.39,6.00),v60,z5,tPen\WObj:=wPaper;
    MoveL Offs(pOrigin,396.12,127.60,6.00),vTravel,z5,tPen\WObj:=wPaper;
    MoveL Offs(pOrigin,396.12,127.60,0.00),v60,z0,tPen\WObj:=wPaper;
    MoveL Offs(pOrigin,394.32,125.80,0.00),v40,fine,tPen\WObj:=wPaper;
    MoveL Offs(pOrigin,394.32,125.80,6.00),v60,z5,tPen\WObj:=wPaper;
    MoveL Offs(pOrigin,386.28,108.28,6.00),vTravel,z5,tPen\WObj:=wPaper;
    MoveL Offs(pOrigin,386.28,108.28,0.00),v60,z0,tPen\WObj:=wPaper;
    MoveL Offs(pOrigin,389.14,105.43,0.00),v40,fine,tPen\WObj:=wPaper;
    MoveL Offs(pOrigin,389.14,105.43,6.00),v60,z5,tPen\WObj:=wPaper;
    MoveL Offs(pOrigin,387.34,105.73,6.00),vTravel,z5,tPen\WObj:=wPaper;
    MoveL Offs(pOrigin,387.34,105.73,0.00),v60,z0,tPen\WObj:=wPaper;
    MoveL Offs(pOrigin,384.49,108.59,0.00),v40,fine,tPen\WObj:=wPaper;
    MoveL Offs(pOrigin,384.49,108.59,6.00),v60,z5,tPen\WObj:=wPaper;
    MoveL Offs(pOrigin,387.36,103.91,6.00),vTravel,z5,tPen\WObj:=wPaper;
    MoveL Offs(pOrigin,387.36,103.91,0.00),v60,z0,tPen\WObj:=wPaper;
    MoveL Offs(pOrigin,386.16,102.70,0.00),v40,fine,tPen\WObj:=wPaper;
    MoveL Offs(pOrigin,386.16,102.70,6.00),v60,z5,tPen\WObj:=wPaper;
    MoveL Offs(pOrigin,388.40,101.96,6.00),vTravel,z5,tPen\WObj:=wPaper;
    MoveL Offs(pOrigin,388.40,101.96,0.00),v60,z0,tPen\WObj:=wPaper;
    MoveL Offs(pOrigin,389.75,103.31,0.00),v40,fine,tPen\WObj:=wPaper;
    MoveL Offs(pOrigin,389.75,103.31,6.00),v60,z5,tPen\WObj:=wPaper;
    MoveL Offs(pOrigin,390.80,101.37,6.00),vTravel,z5,tPen\WObj:=wPaper;
    MoveL Offs(pOrigin,390.80,101.37,0.00),v60,z0,tPen\WObj:=wPaper;
    MoveL Offs(pOrigin,392.00,102.57,0.00),v40,fine,tPen\WObj:=wPaper;
    MoveL Offs(pOrigin,392.00,102.57,6.00),v60,z5,tPen\WObj:=wPaper;
    MoveL Offs(pOrigin,397.98,98.10,6.00),vTravel,z5,tPen\WObj:=wPaper;
    MoveL Offs(pOrigin,397.98,98.10,0.00),v60,z0,tPen\WObj:=wPaper;
    MoveL Offs(pOrigin,398.73,98.85,0.00),v40,fine,tPen\WObj:=wPaper;
    MoveL Offs(pOrigin,398.73,98.85,6.00),v60,z5,tPen\WObj:=wPaper;
    MoveL Offs(pOrigin,409.00,76.26,6.00),vTravel,z5,tPen\WObj:=wPaper;
    MoveL Offs(pOrigin,409.00,76.26,0.00),v60,z0,tPen\WObj:=wPaper;
    MoveL Offs(pOrigin,408.09,75.36,0.00),v40,fine,tPen\WObj:=wPaper;
    MoveL Offs(pOrigin,408.09,75.36,6.00),v60,z5,tPen\WObj:=wPaper;
    MoveL Offs(pOrigin,363.09,100.12,6.00),vTravel,z5,tPen\WObj:=wPaper;
    MoveL Offs(pOrigin,363.09,100.12,0.00),v60,z0,tPen\WObj:=wPaper;
    MoveL Offs(pOrigin,361.74,101.47,0.00),v40,z0,tPen\WObj:=wPaper;
    MoveL Offs(pOrigin,360.84,100.87,0.00),v40,z0,tPen\WObj:=wPaper;
    MoveL Offs(pOrigin,362.34,99.37,0.00),v40,z0,tPen\WObj:=wPaper;
    MoveL Offs(pOrigin,361.77,100.20,0.00),v40,z0,tPen\WObj:=wPaper;
    MoveL Offs(pOrigin,362.20,100.62,0.00),v40,z0,tPen\WObj:=wPaper;
    MoveL Offs(pOrigin,361.77,100.20,0.00),v40,fine,tPen\WObj:=wPaper;
    MoveL Offs(pOrigin,361.77,100.20,6.00),v60,z5,tPen\WObj:=wPaper;
    MoveL Offs(pOrigin,229.60,77.30,6.00),vTravel,z5,tPen\WObj:=wPaper;
    MoveL Offs(pOrigin,229.60,77.30,0.00),v60,z0,tPen\WObj:=wPaper;
    MoveL Offs(pOrigin,228.32,77.30,0.00),v40,z0,tPen\WObj:=wPaper;
    MoveL Offs(pOrigin,228.11,76.25,0.00),v40,z0,tPen\WObj:=wPaper;
    MoveL Offs(pOrigin,229.39,76.25,0.00),v40,z0,tPen\WObj:=wPaper;
    MoveL Offs(pOrigin,229.18,75.19,0.00),v40,z0,tPen\WObj:=wPaper;
    MoveL Offs(pOrigin,227.90,75.19,0.00),v40,z0,tPen\WObj:=wPaper;
    MoveL Offs(pOrigin,227.69,74.14,0.00),v40,z0,tPen\WObj:=wPaper;
    MoveL Offs(pOrigin,228.96,74.14,0.00),v40,z0,tPen\WObj:=wPaper;
    MoveL Offs(pOrigin,228.11,74.06,0.00),v40,z0,tPen\WObj:=wPaper;
    MoveL Offs(pOrigin,228.11,72.79,0.00),v40,z0,tPen\WObj:=wPaper;
    MoveL Offs(pOrigin,227.48,73.08,0.00),v40,z0,tPen\WObj:=wPaper;
    MoveL Offs(pOrigin,228.75,73.08,0.00),v40,z0,tPen\WObj:=wPaper;
    MoveL Offs(pOrigin,228.54,72.02,0.00),v40,z0,tPen\WObj:=wPaper;
    MoveL Offs(pOrigin,227.26,72.02,0.00),v40,fine,tPen\WObj:=wPaper;
    MoveL Offs(pOrigin,227.26,72.02,6.00),v60,z5,tPen\WObj:=wPaper;
    MoveL Offs(pOrigin,229.85,73.56,6.00),vTravel,z5,tPen\WObj:=wPaper;
    MoveL Offs(pOrigin,229.85,73.56,0.00),v60,z0,tPen\WObj:=wPaper;
    MoveL Offs(pOrigin,227.00,76.42,0.00),v40,fine,tPen\WObj:=wPaper;
    MoveL Offs(pOrigin,227.00,76.42,6.00),v60,z5,tPen\WObj:=wPaper;
    MoveL Offs(pOrigin,218.58,84.83,6.00),vTravel,z5,tPen\WObj:=wPaper;
    MoveL Offs(pOrigin,218.58,84.83,0.00),v60,z0,tPen\WObj:=wPaper;
    MoveL Offs(pOrigin,214.82,88.59,0.00),v40,fine,tPen\WObj:=wPaper;
    MoveL Offs(pOrigin,214.82,88.59,6.00),v60,z5,tPen\WObj:=wPaper;
    MoveL Offs(pOrigin,216.21,87.86,6.00),vTravel,z5,tPen\WObj:=wPaper;
    MoveL Offs(pOrigin,216.21,87.86,0.00),v60,z0,tPen\WObj:=wPaper;
    MoveL Offs(pOrigin,217.28,87.86,0.00),v40,z0,tPen\WObj:=wPaper;
    MoveL Offs(pOrigin,217.49,86.81,0.00),v40,z0,tPen\WObj:=wPaper;
    MoveL Offs(pOrigin,216.21,86.81,0.00),v40,fine,tPen\WObj:=wPaper;
    MoveL Offs(pOrigin,216.21,86.81,6.00),v60,z5,tPen\WObj:=wPaper;
    MoveL Offs(pOrigin,216.00,89.98,6.00),vTravel,z5,tPen\WObj:=wPaper;
    MoveL Offs(pOrigin,216.00,89.98,0.00),v60,z0,tPen\WObj:=wPaper;
    MoveL Offs(pOrigin,217.06,89.98,0.00),v40,z0,tPen\WObj:=wPaper;
    MoveL Offs(pOrigin,218.12,89.77,0.00),v40,z0,tPen\WObj:=wPaper;
    MoveL Offs(pOrigin,214.21,93.68,0.00),v40,z0,tPen\WObj:=wPaper;
    MoveL Offs(pOrigin,214.76,94.09,0.00),v40,z0,tPen\WObj:=wPaper;
    MoveL Offs(pOrigin,216.86,96.19,0.00),v40,z0,tPen\WObj:=wPaper;
    MoveL Offs(pOrigin,217.05,96.82,0.00),v40,z0,tPen\WObj:=wPaper;
    MoveL Offs(pOrigin,212.99,100.88,0.00),v40,z0,tPen\WObj:=wPaper;
    MoveL Offs(pOrigin,213.58,100.38,0.00),v40,z0,tPen\WObj:=wPaper;
    MoveL Offs(pOrigin,215.54,102.33,0.00),v40,z0,tPen\WObj:=wPaper;
    MoveL Offs(pOrigin,215.98,102.36,0.00),v40,z0,tPen\WObj:=wPaper;
    MoveL Offs(pOrigin,211.62,106.72,0.00),v40,fine,tPen\WObj:=wPaper;
    MoveL Offs(pOrigin,211.62,106.72,6.00),v60,z5,tPen\WObj:=wPaper;
    MoveL Offs(pOrigin,210.43,106.43,6.00),vTravel,z5,tPen\WObj:=wPaper;
    MoveL Offs(pOrigin,210.43,106.43,0.00),v60,z0,tPen\WObj:=wPaper;
    MoveL Offs(pOrigin,208.32,108.53,0.00),v40,fine,tPen\WObj:=wPaper;
    MoveL Offs(pOrigin,208.32,108.53,6.00),v60,z5,tPen\WObj:=wPaper;
    MoveL Offs(pOrigin,208.48,106.88,6.00),vTravel,z5,tPen\WObj:=wPaper;
    MoveL Offs(pOrigin,208.48,106.88,0.00),v60,z0,tPen\WObj:=wPaper;
    MoveL Offs(pOrigin,210.43,104.93,0.00),v40,fine,tPen\WObj:=wPaper;
    MoveL Offs(pOrigin,210.43,104.93,6.00),v60,z5,tPen\WObj:=wPaper;
    MoveL Offs(pOrigin,210.74,103.13,6.00),vTravel,z5,tPen\WObj:=wPaper;
    MoveL Offs(pOrigin,210.74,103.13,0.00),v60,z0,tPen\WObj:=wPaper;
    MoveL Offs(pOrigin,208.48,105.38,0.00),v40,fine,tPen\WObj:=wPaper;
  ENDPROC

  PROC DrawPart275()
    MoveL Offs(pOrigin,208.48,105.38,6.00),v60,z5,tPen\WObj:=wPaper;
    MoveL Offs(pOrigin,208.64,103.73,6.00),vTravel,z5,tPen\WObj:=wPaper;
    MoveL Offs(pOrigin,208.64,103.73,0.00),v60,z0,tPen\WObj:=wPaper;
    MoveL Offs(pOrigin,210.74,101.63,0.00),v40,fine,tPen\WObj:=wPaper;
    MoveL Offs(pOrigin,210.74,101.63,6.00),v60,z5,tPen\WObj:=wPaper;
    MoveL Offs(pOrigin,210.90,99.98,6.00),vTravel,z5,tPen\WObj:=wPaper;
    MoveL Offs(pOrigin,210.90,99.98,0.00),v60,z0,tPen\WObj:=wPaper;
    MoveL Offs(pOrigin,208.94,101.94,0.00),v40,fine,tPen\WObj:=wPaper;
    MoveL Offs(pOrigin,208.94,101.94,6.00),v60,z5,tPen\WObj:=wPaper;
    MoveL Offs(pOrigin,209.10,100.29,6.00),vTravel,z5,tPen\WObj:=wPaper;
    MoveL Offs(pOrigin,209.10,100.29,0.00),v60,z0,tPen\WObj:=wPaper;
    MoveL Offs(pOrigin,210.90,98.49,0.00),v40,fine,tPen\WObj:=wPaper;
    MoveL Offs(pOrigin,210.90,98.49,6.00),v60,z5,tPen\WObj:=wPaper;
    MoveL Offs(pOrigin,210.90,96.99,6.00),vTravel,z5,tPen\WObj:=wPaper;
    MoveL Offs(pOrigin,210.90,96.99,0.00),v60,z0,tPen\WObj:=wPaper;
    MoveL Offs(pOrigin,209.40,98.49,0.00),v40,fine,tPen\WObj:=wPaper;
    MoveL Offs(pOrigin,209.40,98.49,6.00),v60,z5,tPen\WObj:=wPaper;
    MoveL Offs(pOrigin,209.86,96.54,6.00),vTravel,z5,tPen\WObj:=wPaper;
    MoveL Offs(pOrigin,209.86,96.54,0.00),v60,z0,tPen\WObj:=wPaper;
    MoveL Offs(pOrigin,210.91,95.49,0.00),v40,fine,tPen\WObj:=wPaper;
    MoveL Offs(pOrigin,210.91,95.49,6.00),v60,z5,tPen\WObj:=wPaper;
    MoveL Offs(pOrigin,214.94,96.31,6.00),vTravel,z5,tPen\WObj:=wPaper;
    MoveL Offs(pOrigin,214.94,96.31,0.00),v60,z0,tPen\WObj:=wPaper;
    MoveL Offs(pOrigin,216.21,96.31,0.00),v40,z0,tPen\WObj:=wPaper;
    MoveL Offs(pOrigin,216.42,95.26,0.00),v40,z0,tPen\WObj:=wPaper;
    MoveL Offs(pOrigin,215.15,95.26,0.00),v40,z0,tPen\WObj:=wPaper;
    MoveL Offs(pOrigin,215.36,94.20,0.00),v40,z0,tPen\WObj:=wPaper;
    MoveL Offs(pOrigin,216.42,94.20,0.00),v40,z0,tPen\WObj:=wPaper;
    MoveL Offs(pOrigin,216.64,93.14,0.00),v40,z0,tPen\WObj:=wPaper;
    MoveL Offs(pOrigin,215.58,93.14,0.00),v40,fine,tPen\WObj:=wPaper;
    MoveL Offs(pOrigin,215.58,93.14,6.00),v60,z5,tPen\WObj:=wPaper;
    MoveL Offs(pOrigin,215.79,91.03,6.00),vTravel,z5,tPen\WObj:=wPaper;
    MoveL Offs(pOrigin,215.79,91.03,0.00),v60,z0,tPen\WObj:=wPaper;
    MoveL Offs(pOrigin,216.85,91.03,0.00),v40,fine,tPen\WObj:=wPaper;
    MoveL Offs(pOrigin,216.85,91.03,6.00),v60,z5,tPen\WObj:=wPaper;
    MoveL Offs(pOrigin,210.69,91.06,6.00),vTravel,z5,tPen\WObj:=wPaper;
    MoveL Offs(pOrigin,210.69,91.06,0.00),v60,z0,tPen\WObj:=wPaper;
    MoveL Offs(pOrigin,210.90,91.49,0.00),v40,z0,tPen\WObj:=wPaper;
    MoveL Offs(pOrigin,209.62,105.51,0.00),v40,z0,tPen\WObj:=wPaper;
    MoveL Offs(pOrigin,207.93,119.32,0.00),v40,z0,tPen\WObj:=wPaper;
    MoveL Offs(pOrigin,208.14,120.60,0.00),v40,z0,tPen\WObj:=wPaper;
    MoveL Offs(pOrigin,208.35,120.60,0.00),v40,z0,tPen\WObj:=wPaper;
    MoveL Offs(pOrigin,210.26,120.60,0.00),v40,z0,tPen\WObj:=wPaper;
    MoveL Offs(pOrigin,210.65,121.34,0.00),v40,z0,tPen\WObj:=wPaper;
    MoveL Offs(pOrigin,207.49,118.18,0.00),v40,fine,tPen\WObj:=wPaper;
    MoveL Offs(pOrigin,207.49,118.18,6.00),v60,z5,tPen\WObj:=wPaper;
    MoveL Offs(pOrigin,207.50,119.68,6.00),vTravel,z5,tPen\WObj:=wPaper;
    MoveL Offs(pOrigin,207.50,119.68,0.00),v60,z0,tPen\WObj:=wPaper;
    MoveL Offs(pOrigin,210.35,122.54,0.00),v40,z0,tPen\WObj:=wPaper;
    MoveL Offs(pOrigin,210.83,122.45,0.00),v40,z0,tPen\WObj:=wPaper;
    MoveL Offs(pOrigin,205.42,127.86,0.00),v40,fine,tPen\WObj:=wPaper;
    MoveL Offs(pOrigin,205.42,127.86,6.00),v60,z5,tPen\WObj:=wPaper;
    MoveL Offs(pOrigin,206.65,127.99,6.00),vTravel,z5,tPen\WObj:=wPaper;
    MoveL Offs(pOrigin,206.65,127.99,0.00),v60,z0,tPen\WObj:=wPaper;
    MoveL Offs(pOrigin,208.35,127.99,0.00),v40,z0,tPen\WObj:=wPaper;
    MoveL Offs(pOrigin,208.05,126.98,0.00),v40,z0,tPen\WObj:=wPaper;
    MoveL Offs(pOrigin,208.05,123.36,0.00),v40,z0,tPen\WObj:=wPaper;
    MoveL Offs(pOrigin,207.71,122.71,0.00),v40,z0,tPen\WObj:=wPaper;
    MoveL Offs(pOrigin,209.84,122.71,0.00),v40,z0,tPen\WObj:=wPaper;
    MoveL Offs(pOrigin,209.10,123.15,0.00),v40,z0,tPen\WObj:=wPaper;
    MoveL Offs(pOrigin,209.10,121.24,0.00),v40,z0,tPen\WObj:=wPaper;
    MoveL Offs(pOrigin,210.05,121.66,0.00),v40,z0,tPen\WObj:=wPaper;
    MoveL Offs(pOrigin,207.92,121.66,0.00),v40,fine,tPen\WObj:=wPaper;
    MoveL Offs(pOrigin,207.92,121.66,6.00),v60,z5,tPen\WObj:=wPaper;
    MoveL Offs(pOrigin,208.78,119.54,6.00),vTravel,z5,tPen\WObj:=wPaper;
    MoveL Offs(pOrigin,208.78,119.54,0.00),v60,z0,tPen\WObj:=wPaper;
    MoveL Offs(pOrigin,210.69,119.54,0.00),v40,fine,tPen\WObj:=wPaper;
    MoveL Offs(pOrigin,210.69,119.54,6.00),v60,z5,tPen\WObj:=wPaper;
    MoveL Offs(pOrigin,210.22,124.55,6.00),vTravel,z5,tPen\WObj:=wPaper;
    MoveL Offs(pOrigin,210.22,124.55,0.00),v60,z0,tPen\WObj:=wPaper;
    MoveL Offs(pOrigin,205.26,129.51,0.00),v40,fine,tPen\WObj:=wPaper;
    MoveL Offs(pOrigin,205.26,129.51,6.00),v60,z5,tPen\WObj:=wPaper;
    MoveL Offs(pOrigin,204.81,131.46,6.00),vTravel,z5,tPen\WObj:=wPaper;
    MoveL Offs(pOrigin,204.81,131.46,0.00),v60,z0,tPen\WObj:=wPaper;
    MoveL Offs(pOrigin,209.62,126.65,0.00),v40,fine,tPen\WObj:=wPaper;
    MoveL Offs(pOrigin,209.62,126.65,6.00),v60,z5,tPen\WObj:=wPaper;
    MoveL Offs(pOrigin,208.25,131.00,6.00),vTravel,z5,tPen\WObj:=wPaper;
    MoveL Offs(pOrigin,208.25,131.00,0.00),v60,z0,tPen\WObj:=wPaper;
    MoveL Offs(pOrigin,203.45,135.81,0.00),v40,fine,tPen\WObj:=wPaper;
    MoveL Offs(pOrigin,203.45,135.81,6.00),v60,z5,tPen\WObj:=wPaper;
    MoveL Offs(pOrigin,204.52,136.44,6.00),vTravel,z5,tPen\WObj:=wPaper;
    MoveL Offs(pOrigin,204.52,136.44,0.00),v60,z0,tPen\WObj:=wPaper;
    MoveL Offs(pOrigin,205.80,136.44,0.00),v40,z0,tPen\WObj:=wPaper;
    MoveL Offs(pOrigin,206.35,136.46,0.00),v40,z0,tPen\WObj:=wPaper;
    MoveL Offs(pOrigin,204.40,134.50,0.00),v40,z0,tPen\WObj:=wPaper;
    MoveL Offs(pOrigin,205.16,134.33,0.00),v40,z0,tPen\WObj:=wPaper;
    MoveL Offs(pOrigin,206.44,134.33,0.00),v40,z0,tPen\WObj:=wPaper;
    MoveL Offs(pOrigin,207.09,134.21,0.00),v40,z0,tPen\WObj:=wPaper;
    MoveL Offs(pOrigin,205.29,132.41,0.00),v40,z0,tPen\WObj:=wPaper;
    MoveL Offs(pOrigin,205.80,132.22,0.00),v40,z0,tPen\WObj:=wPaper;
    MoveL Offs(pOrigin,207.08,132.22,0.00),v40,z0,tPen\WObj:=wPaper;
    MoveL Offs(pOrigin,206.65,133.27,0.00),v40,z0,tPen\WObj:=wPaper;
    MoveL Offs(pOrigin,205.38,133.27,0.00),v40,fine,tPen\WObj:=wPaper;
    MoveL Offs(pOrigin,205.38,133.27,6.00),v60,z5,tPen\WObj:=wPaper;
    MoveL Offs(pOrigin,207.19,135.05,6.00),vTravel,z5,tPen\WObj:=wPaper;
    MoveL Offs(pOrigin,207.19,135.05,0.00),v60,z0,tPen\WObj:=wPaper;
    MoveL Offs(pOrigin,202.38,139.86,0.00),v40,fine,tPen\WObj:=wPaper;
    MoveL Offs(pOrigin,202.38,139.86,6.00),v60,z5,tPen\WObj:=wPaper;
    MoveL Offs(pOrigin,201.78,141.95,6.00),vTravel,z5,tPen\WObj:=wPaper;
    MoveL Offs(pOrigin,201.78,141.95,0.00),v60,z0,tPen\WObj:=wPaper;
    MoveL Offs(pOrigin,206.59,137.15,0.00),v40,fine,tPen\WObj:=wPaper;
    MoveL Offs(pOrigin,206.59,137.15,6.00),v60,z5,tPen\WObj:=wPaper;
    MoveL Offs(pOrigin,203.68,143.83,6.00),vTravel,z5,tPen\WObj:=wPaper;
    MoveL Offs(pOrigin,203.68,143.83,0.00),v60,z0,tPen\WObj:=wPaper;
    MoveL Offs(pOrigin,202.61,143.83,0.00),v40,z0,tPen\WObj:=wPaper;
    MoveL Offs(pOrigin,202.19,144.89,0.00),v40,z0,tPen\WObj:=wPaper;
    MoveL Offs(pOrigin,203.46,144.89,0.00),v40,fine,tPen\WObj:=wPaper;
    MoveL Offs(pOrigin,203.46,144.89,6.00),v60,z5,tPen\WObj:=wPaper;
    MoveL Offs(pOrigin,201.12,153.34,6.00),vTravel,z5,tPen\WObj:=wPaper;
    MoveL Offs(pOrigin,201.12,153.34,0.00),v60,z0,tPen\WObj:=wPaper;
    MoveL Offs(pOrigin,200.06,153.34,0.00),v40,fine,tPen\WObj:=wPaper;
    MoveL Offs(pOrigin,200.06,153.34,6.00),v60,z5,tPen\WObj:=wPaper;
    MoveL Offs(pOrigin,229.60,147.00,6.00),vTravel,z5,tPen\WObj:=wPaper;
    MoveL Offs(pOrigin,229.60,147.00,0.00),v60,z0,tPen\WObj:=wPaper;
    MoveL Offs(pOrigin,230.66,147.00,0.00),v40,fine,tPen\WObj:=wPaper;
    MoveL Offs(pOrigin,230.66,147.00,6.00),v60,z5,tPen\WObj:=wPaper;
    MoveL Offs(pOrigin,230.88,144.89,6.00),vTravel,z5,tPen\WObj:=wPaper;
    MoveL Offs(pOrigin,230.88,144.89,0.00),v60,z0,tPen\WObj:=wPaper;
    MoveL Offs(pOrigin,229.81,144.89,0.00),v40,fine,tPen\WObj:=wPaper;
    MoveL Offs(pOrigin,229.81,144.89,6.00),v60,z5,tPen\WObj:=wPaper;
  ENDPROC

